    |   movel([0.131422, -1.358046, -2.590069, -0.764274, 1.570796, 1.702219],accel_mss,speed_ms,0,blend_radius_m)
    |   movel([0.131217, -1.358381, -2.589844, -0.764164, 1.570796, 1.702013],accel_mss,speed_ms,0,blend_radius_m)
    |   movel([0.131469, -1.358672, -2.589647, -0.764069, 1.570796, 1.702265],accel_mss,speed_ms,0,blend_radius_m)
    |   movel([0.131675, -1.358796, -2.589564, -0.764029, 1.570796, 1.702471],accel_mss,speed_ms,0,blend_radius_m)
    |   movel([0.131656, -1.359066, -2.589382, -0.763941, 1.570796, 1.702453],accel_mss,speed_ms,0,blend_radius_m)
    |   movel([0.131428, -1.359319, -2.589211, -0.763858, 1.570796, 1.702225],accel_mss,speed_ms,0,blend_radius_m)
    |   movel([0.131132, -1.359619, -2.589009, -0.763761, 1.570796, 1.701929],accel_mss,speed_ms,0,blend_radius_m)
    |   movel([0.127085, -1.360149, -2.588651, -0.763589, 1.570796, 1.697882],accel_mss,speed_ms,0,blend_radius_m)
    |   movel([0.125499, -1.360363, -2.588507, -0.763519, 1.570796, 1.696296],accel_mss,speed_ms,0,blend_radius_m)
    |   movel([0.124079, -1.360556, -2.588376, -0.763457, 1.570796, 1.694875],accel_mss,speed_ms,0,blend_radius_m)
    |   movel([0.122882, -1.360722, -2.588264, -0.763403, 1.570796, 1.693678],accel_mss,speed_ms,0,blend_radius_m)
    |   movel([0.122534, -1.360775, -2.588228, -0.763386, 1.570796, 1.693331],accel_mss,speed_ms,0,blend_radius_m)
    |   movel([0.122267, -1.360818, -2.588199, -0.763372, 1.570796, 1.693063],accel_mss,speed_ms,0,blend_radius_m)
    |   movel([0.121847, -1.360878, -2.588158, -0.763353, 1.570796, 1.692643],accel_mss,speed_ms,0,blend_radius_m)
    |   movel([0.121369, -1.360945, -2.588113, -0.763331, 1.570796, 1.692165],accel_mss,speed_ms,0,blend_radius_m)
    |   movel([0.120899, -1.361009, -2.588070, -0.763311, 1.570796, 1.691695],accel_mss,speed_ms,0,blend_radius_m)
    |   movel([0.120401, -1.361077, -2.588023, -0.763288, 1.570796, 1.691197],accel_mss,speed_ms,0,blend_radius_m)
    |   movel([0.119840, -1.361153, -2.587972, -0.763264, 1.570796, 1.690636],accel_mss,speed_ms,0,blend_radius_m)
    |   movel([0.119304, -1.361228, -2.587921, -0.763240, 1.570796, 1.690101],accel_mss,speed_ms,0,blend_radius_m)
    |   movel([0.118887, -1.361287, -2.587881, -0.763221, 1.570796, 1.689683],accel_mss,speed_ms,0,blend_radius_m)
    |   movel([0.118469, -1.361347, -2.587840, -0.763201, 1.570796, 1.689265],accel_mss,speed_ms,0,blend_radius_m)
    |   movel([0.117933, -1.361421, -2.587790, -0.763178, 1.570796, 1.688730],accel_mss,speed_ms,0,blend_radius_m)
    |   movel([0.117372, -1.361500, -2.587737, -0.763152, 1.570796, 1.688169],accel_mss,speed_ms,0,blend_radius_m)
    |   movel([0.116874, -1.361570, -2.587689, -0.763129, 1.570796, 1.687671],accel_mss,speed_ms,0,blend_radius_m)
    |   movel([0.114544, -1.361902, -2.587464, -0.763022, 1.570796, 1.685341],accel_mss,speed_ms,0,blend_radius_m)
    |   movel([0.111844, -1.362308, -2.587189, -0.762892, 1.570796, 1.682641],accel_mss,speed_ms,0,blend_radius_m)
    |   movel([0.109120, -1.362733, -2.586901, -0.762756, 1.570796, 1.679916],accel_mss,speed_ms,0,blend_radius_m)
    |   movel([0.108772, -1.362809, -2.586848, -0.762731, 1.570796, 1.679568],accel_mss,speed_ms,0,blend_radius_m)
    |   movel([0.108514, -1.362574, -2.587008, -0.762807, 1.570796, 1.679311],accel_mss,speed_ms,0,blend_radius_m)
    |   movel([0.108672, -1.362243, -2.587233, -0.762913, 1.570796, 1.679468],accel_mss,speed_ms,0,blend_radius_m)
    |   movel([0.108981, -1.361907, -2.587461, -0.763021, 1.570796, 1.679777],accel_mss,speed_ms,0,blend_radius_m)
    |   movel([0.109311, -1.361648, -2.587636, -0.763104, 1.570796, 1.680107],accel_mss,speed_ms,0,blend_radius_m)
    |   movel([0.109605, -1.361472, -2.587756, -0.763161, 1.570796, 1.680401],accel_mss,speed_ms,0,blend_radius_m)
    |   movel([0.109666, -1.361181, -2.587953, -0.763255, 1.570796, 1.680463],accel_mss,speed_ms,0,blend_radius_m)
    |   movel([0.109470, -1.361072, -2.588027, -0.763290, 1.570796, 1.680266],accel_mss,speed_ms,0,blend_radius_m)
    |   movel([0.109530, -1.360833, -2.588189, -0.763367, 1.570796, 1.680326],accel_mss,speed_ms,0,blend_radius_m)
    |   movel([0.109705, -1.360578, -2.588361, -0.763450, 1.570796, 1.680502],accel_mss,speed_ms,0,blend_radius_m)
    |   movel([0.109652, -1.360212, -2.588608, -0.763568, 1.570796, 1.680449],accel_mss,speed_ms,0,blend_radius_m)
    |   movel([0.109837, -1.359966, -2.588775, -0.763648, 1.570796, 1.680633],accel_mss,speed_ms,0,blend_radius_m)
    |   movel([0.109967, -1.359524, -2.589073, -0.763792, 1.570796, 1.680764],accel_mss,speed_ms,0,blend_radius_m)
    |   movel([0.110006, -1.359241, -2.589264, -0.763884, 1.570796, 1.680802],accel_mss,speed_ms,0,blend_radius_m)
    |   movel([0.110093, -1.358670, -2.589649, -0.764070, 1.570796, 1.680889],accel_mss,speed_ms,0,blend_radius_m)
    |   movel([0.110206, -1.358204, -2.589963, -0.764222, 1.570796, 1.681003],accel_mss,speed_ms,0,blend_radius_m)
    |   movel([0.110408, -1.357592, -2.590375, -0.764422, 1.570796, 1.681205],accel_mss,speed_ms,0,blend_radius_m)
    |   movel([0.110894, -1.356270, -2.591262, -0.764857, 1.570796, 1.681691],accel_mss,speed_ms,0,blend_radius_m)
    |   movel([0.111101, -1.355724, -2.591628, -0.765037, 1.570796, 1.681897],accel_mss,speed_ms,0,blend_radius_m)
    |   movel([0.111293, -1.355253, -2.591943, -0.765193, 1.570796, 1.682089],accel_mss,speed_ms,0,blend_radius_m)
    |   movel([0.111466, -1.354854, -2.592210, -0.765325, 1.570796, 1.682262],accel_mss,speed_ms,0,blend_radius_m)
    |   movel([0.111570, -1.354589, -2.592387, -0.765413, 1.570796, 1.682366],accel_mss,speed_ms,0,blend_radius_m)
    |   movel([0.111744, -1.354339, -2.592554, -0.765496, 1.570796, 1.682540],accel_mss,speed_ms,0,blend_radius_m)
    |   movel([0.111777, -1.353985, -2.592790, -0.765614, 1.570796, 1.682573],accel_mss,speed_ms,0,blend_radius_m)
    |   movel([0.112301, -1.352877, -2.593529, -0.765984, 1.570796, 1.683097],accel_mss,speed_ms,0,blend_radius_m)
    |   movel([0.112851, -1.351791, -2.594251, -0.766348, 1.570796, 1.683647],accel_mss,speed_ms,0,blend_radius_m)
    |   movel([0.113284, -1.351070, -2.594729, -0.766590, 1.570796, 1.684081],accel_mss,speed_ms,0,blend_radius_m)
    |   movel([0.113462, -1.350817, -2.594896, -0.766675, 1.570796, 1.684258],accel_mss,speed_ms,0,blend_radius_m)
    |   movel([0.113667, -1.350551, -2.595073, -0.766765, 1.570796, 1.684463],accel_mss,speed_ms,0,blend_radius_m)
    |   movel([0.113872, -1.350302, -2.595238, -0.766849, 1.570796, 1.684668],accel_mss,speed_ms,0,blend_radius_m)
    |   movel([0.114255, -1.349877, -2.595519, -0.766993, 1.570796, 1.685052],accel_mss,speed_ms,0,blend_radius_m)
    |   movel([0.114419, -1.349522, -2.595753, -0.767113, 1.570796, 1.685216],accel_mss,speed_ms,0,blend_radius_m)
    |   movel([0.114172, -1.349540, -2.595742, -0.767107, 1.570796, 1.684968],accel_mss,speed_ms,0,blend_radius_m)
    |   movel([0.113906, -1.349563, -2.595727, -0.767099, 1.570796, 1.684702],accel_mss,speed_ms,0,blend_radius_m)
    |   movel([0.113638, -1.349488, -2.595776, -0.767125, 1.570796, 1.684434],accel_mss,speed_ms,0,blend_radius_m)
    |   movel([0.113581, -1.349115, -2.596022, -0.767251, 1.570796, 1.684377],accel_mss,speed_ms,0,blend_radius_m)
    |   movel([0.113640, -1.348716, -2.596286, -0.767387, 1.570796, 1.684437],accel_mss,speed_ms,0,blend_radius_m)
    |   movel([0.113813, -1.348451, -2.596461, -0.767477, 1.570796, 1.684609],accel_mss,speed_ms,0,blend_radius_m)
    |   movel([0.114104, -1.348214, -2.596617, -0.767558, 1.570796, 1.684901],accel_mss,speed_ms,0,blend_radius_m)
    |   movel([0.114427, -1.348012, -2.596750, -0.767627, 1.570796, 1.685223],accel_mss,speed_ms,0,blend_radius_m)
    |   movel([0.114780, -1.347843, -2.596862, -0.767685, 1.570796, 1.685576],accel_mss,speed_ms,0,blend_radius_m)
    |   movel([0.115153, -1.347715, -2.596946, -0.767728, 1.570796, 1.685950],accel_mss,speed_ms,0,blend_radius_m)
    |   movel([0.115538, -1.347574, -2.597038, -0.767776, 1.570796, 1.686334],accel_mss,speed_ms,0,blend_radius_m)
    |   movel([0.116178, -1.347179, -2.597299, -0.767912, 1.570796, 1.686974],accel_mss,speed_ms,0,blend_radius_m)
    |   movel([0.118416, -1.346430, -2.597791, -0.768168, 1.570796, 1.689213],accel_mss,speed_ms,0,blend_radius_m)
    |   movel([0.120675, -1.345699, -2.598271, -0.768420, 1.570796, 1.691471],accel_mss,speed_ms,0,blend_radius_m)
    |   movel([0.120996, -1.345719, -2.598257, -0.768413, 1.570796, 1.691792],accel_mss,speed_ms,0,blend_radius_m)
    |   movel([0.121352, -1.345738, -2.598245, -0.768406, 1.570796, 1.692148],accel_mss,speed_ms,0,blend_radius_m)
    |   movel([0.121691, -1.345520, -2.598388, -0.768481, 1.570796, 1.692487],accel_mss,speed_ms,0,blend_radius_m)
    |   movel([0.121589, -1.345278, -2.598546, -0.768565, 1.570796, 1.692385],accel_mss,speed_ms,0,blend_radius_m)
    |   movel([0.121500, -1.344976, -2.598744, -0.768669, 1.570796, 1.692296],accel_mss,speed_ms,0,blend_radius_m)
    |   movel([0.121695, -1.344748, -2.598893, -0.768748, 1.570796, 1.692491],accel_mss,speed_ms,0,blend_radius_m)
    |   movel([0.122038, -1.344499, -2.599056, -0.768834, 1.570796, 1.692835],accel_mss,speed_ms,0,blend_radius_m)
    |   movel([0.122298, -1.344313, -2.599178, -0.768898, 1.570796, 1.693094],accel_mss,speed_ms,0,blend_radius_m)
    |   movel([0.122428, -1.344051, -2.599349, -0.768989, 1.570796, 1.693224],accel_mss,speed_ms,0,blend_radius_m)
    |   movel([0.122134, -1.344045, -2.599353, -0.768991, 1.570796, 1.692931],accel_mss,speed_ms,0,blend_radius_m)
    |   movel([0.121865, -1.344049, -2.599350, -0.768989, 1.570796, 1.692661],accel_mss,speed_ms,0,blend_radius_m)
    |   movel([0.121926, -1.343536, -2.599686, -0.769168, 1.570796, 1.692722],accel_mss,speed_ms,0,blend_radius_m)
    |   movel([0.122108, -1.342970, -2.600055, -0.769365, 1.570796, 1.692904],accel_mss,speed_ms,0,blend_radius_m)
    |   movel([0.122198, -1.342705, -2.600227, -0.769457, 1.570796, 1.692994],accel_mss,speed_ms,0,blend_radius_m)
    |   movel([0.122277, -1.342458, -2.600388, -0.769543, 1.570796, 1.693074],accel_mss,speed_ms,0,blend_radius_m)
    |   movel([0.122367, -1.342155, -2.600585, -0.769649, 1.570796, 1.693164],accel_mss,speed_ms,0,blend_radius_m)
    |   movel([0.122577, -1.341845, -2.600787, -0.769757, 1.570796, 1.693373],accel_mss,speed_ms,0,blend_radius_m)
    |   movel([0.122789, -1.341589, -2.600953, -0.769846, 1.570796, 1.693585],accel_mss,speed_ms,0,blend_radius_m)
    |   movel([0.123034, -1.341314, -2.601133, -0.769943, 1.570796, 1.693831],accel_mss,speed_ms,0,blend_radius_m)
    |   movel([0.123671, -1.340622, -2.601581, -0.770185, 1.570796, 1.694467],accel_mss,speed_ms,0,blend_radius_m)
    |   movel([0.124629, -1.340427, -2.601708, -0.770254, 1.570796, 1.695426],accel_mss,speed_ms,0,blend_radius_m)
    |   movel([0.125882, -1.340203, -2.601853, -0.770333, 1.570796, 1.696678],accel_mss,speed_ms,0,blend_radius_m)
    |   movel([0.127200, -1.340030, -2.601965, -0.770394, 1.570796, 1.697996],accel_mss,speed_ms,0,blend_radius_m)
    |   movel([0.128376, -1.339917, -2.602039, -0.770434, 1.570796, 1.699172],accel_mss,speed_ms,0,blend_radius_m)
    |   movel([0.128803, -1.339961, -2.602010, -0.770418, 1.570796, 1.699599],accel_mss,speed_ms,0,blend_radius_m)
    |   movel([0.129089, -1.340087, -2.601928, -0.770374, 1.570796, 1.699886],accel_mss,speed_ms,0,blend_radius_m)
    |   movel([0.129309, -1.340254, -2.601820, -0.770315, 1.570796, 1.700106],accel_mss,speed_ms,0,blend_radius_m)
    |   movel([0.129435, -1.340429, -2.601707, -0.770253, 1.570796, 1.700231],accel_mss,speed_ms,0,blend_radius_m)
    |   movel([0.129396, -1.340689, -2.601538, -0.770162, 1.570796, 1.700193],accel_mss,speed_ms,0,blend_radius_m)
    |   movel([0.129524, -1.340866, -2.601423, -0.770100, 1.570796, 1.700320],accel_mss,speed_ms,0,blend_radius_m)
    |   movel([0.129472, -1.341183, -2.601217, -0.769989, 1.570796, 1.700269],accel_mss,speed_ms,0,blend_radius_m)
    |   movel([0.129264, -1.341421, -2.601063, -0.769905, 1.570796, 1.700060],accel_mss,speed_ms,0,blend_radius_m)
    |   movel([0.129247, -1.341706, -2.600878, -0.769806, 1.570796, 1.700043],accel_mss,speed_ms,0,blend_radius_m)
    |   movel([0.129226, -1.342103, -2.600619, -0.769667, 1.570796, 1.700023],accel_mss,speed_ms,0,blend_radius_m)
    |   movel([0.129118, -1.342564, -2.600319, -0.769506, 1.570796, 1.699915],accel_mss,speed_ms,0,blend_radius_m)
    |   movel([0.128966, -1.342955, -2.600064, -0.769370, 1.570796, 1.699762],accel_mss,speed_ms,0,blend_radius_m)
    |   movel([0.128664, -1.343092, -2.599975, -0.769322, 1.570796, 1.699461],accel_mss,speed_ms,0,blend_radius_m)
    |   movel([0.128382, -1.343292, -2.599845, -0.769252, 1.570796, 1.699178],accel_mss,speed_ms,0,blend_radius_m)
    |   movel([0.128379, -1.343588, -2.599652, -0.769150, 1.570796, 1.699175],accel_mss,speed_ms,0,blend_radius_m)
    |   movel([0.128483, -1.343834, -2.599491, -0.769064, 1.570796, 1.699279],accel_mss,speed_ms,0,blend_radius_m)
    |   movel([0.128519, -1.344124, -2.599301, -0.768964, 1.570796, 1.699315],accel_mss,speed_ms,0,blend_radius_m)
    |   movel([0.128237, -1.344388, -2.599129, -0.768872, 1.570796, 1.699033],accel_mss,speed_ms,0,blend_radius_m)
    |   movel([0.128151, -1.344682, -2.598937, -0.768771, 1.570796, 1.698948],accel_mss,speed_ms,0,blend_radius_m)
    |   movel([0.128545, -1.344644, -2.598961, -0.768784, 1.570796, 1.699342],accel_mss,speed_ms,0,blend_radius_m)
    |   movel([0.129417, -1.344531, -2.599035, -0.768823, 1.570796, 1.700213],accel_mss,speed_ms,0,blend_radius_m)
    |   movel([0.130216, -1.344512, -2.599048, -0.768829, 1.570796, 1.701013],accel_mss,speed_ms,0,blend_radius_m)
    |   movel([0.130962, -1.344536, -2.599032, -0.768821, 1.570796, 1.701758],accel_mss,speed_ms,0,blend_radius_m)
    |   movel([0.131239, -1.344625, -2.598974, -0.768790, 1.570796, 1.702036],accel_mss,speed_ms,0,blend_radius_m)
    |   movel([0.131699, -1.344650, -2.598957, -0.768781, 1.570796, 1.702495],accel_mss,speed_ms,0,blend_radius_m)
    |   movel([0.132047, -1.344467, -2.599077, -0.768845, 1.570796, 1.702843],accel_mss,speed_ms,0,blend_radius_m)
    |   movel([0.131918, -1.344291, -2.599192, -0.768906, 1.570796, 1.702714],accel_mss,speed_ms,0,blend_radius_m)
    |   movel([0.131651, -1.344100, -2.599317, -0.768972, 1.570796, 1.702447],accel_mss,speed_ms,0,blend_radius_m)
    |   movel([0.132106, -1.343657, -2.599607, -0.769126, 1.570796, 1.702902],accel_mss,speed_ms,0,blend_radius_m)
    |   movel([0.132430, -1.343451, -2.599741, -0.769197, 1.570796, 1.703227],accel_mss,speed_ms,0,blend_radius_m)
    |   movel([0.132572, -1.343210, -2.599898, -0.769281, 1.570796, 1.703368],accel_mss,speed_ms,0,blend_radius_m)
    |   movel([0.132296, -1.343074, -2.599987, -0.769328, 1.570796, 1.703093],accel_mss,speed_ms,0,blend_radius_m)
    |   movel([0.132431, -1.342597, -2.600298, -0.769494, 1.570796, 1.703227],accel_mss,speed_ms,0,blend_radius_m)
    |   movel([0.132665, -1.342355, -2.600455, -0.769579, 1.570796, 1.703462],accel_mss,speed_ms,0,blend_radius_m)
    |   movel([0.133142, -1.342023, -2.600671, -0.769695, 1.570796, 1.703938],accel_mss,speed_ms,0,blend_radius_m)
    |   movel([0.133515, -1.341866, -2.600774, -0.769750, 1.570796, 1.704311],accel_mss,speed_ms,0,blend_radius_m)
    |   movel([0.133874, -1.341846, -2.600787, -0.769757, 1.570796, 1.704671],accel_mss,speed_ms,0,blend_radius_m)
    |   movel([0.134312, -1.341959, -2.600713, -0.769717, 1.570796, 1.705108],accel_mss,speed_ms,0,blend_radius_m)
    |   movel([0.134537, -1.342047, -2.600656, -0.769686, 1.570796, 1.705333],accel_mss,speed_ms,0,blend_radius_m)
    |   movel([0.134724, -1.342134, -2.600599, -0.769656, 1.570796, 1.705520],accel_mss,speed_ms,0,blend_radius_m)
    |   movel([0.134889, -1.342254, -2.600521, -0.769614, 1.570796, 1.705685],accel_mss,speed_ms,0,blend_radius_m)
    |   movel([0.135058, -1.342462, -2.600386, -0.769541, 1.570796, 1.705854],accel_mss,speed_ms,0,blend_radius_m)
    |   movel([0.135120, -1.342790, -2.600172, -0.769427, 1.570796, 1.705917],accel_mss,speed_ms,0,blend_radius_m)
    |   movel([0.134596, -1.343303, -2.599837, -0.769249, 1.570796, 1.705392],accel_mss,speed_ms,0,blend_radius_m)
    |   movel([0.134152, -1.343634, -2.599621, -0.769134, 1.570796, 1.704948],accel_mss,speed_ms,0,blend_radius_m)
    |   movel([0.134394, -1.343806, -2.599509, -0.769074, 1.570796, 1.705190],accel_mss,speed_ms,0,blend_radius_m)
    |   movel([0.134638, -1.343980, -2.599395, -0.769013, 1.570796, 1.705434],accel_mss,speed_ms,0,blend_radius_m)
    |   movel([0.134303, -1.344283, -2.599197, -0.768908, 1.570796, 1.705100],accel_mss,speed_ms,0,blend_radius_m)
    |   movel([0.133995, -1.344518, -2.599044, -0.768827, 1.570796, 1.704791],accel_mss,speed_ms,0,blend_radius_m)
    |   movel([0.133724, -1.344655, -2.598954, -0.768780, 1.570796, 1.704520],accel_mss,speed_ms,0,blend_radius_m)
    |   movel([0.133806, -1.344937, -2.598770, -0.768682, 1.570796, 1.704602],accel_mss,speed_ms,0,blend_radius_m)
    |   movel([0.134102, -1.344945, -2.598764, -0.768679, 1.570796, 1.704899],accel_mss,speed_ms,0,blend_radius_m)
    |   movel([0.134405, -1.344992, -2.598733, -0.768663, 1.570796, 1.705202],accel_mss,speed_ms,0,blend_radius_m)
    |   movel([0.134632, -1.345146, -2.598633, -0.768610, 1.570796, 1.705428],accel_mss,speed_ms,0,blend_radius_m)
    |   movel([0.134781, -1.345283, -2.598543, -0.768563, 1.570796, 1.705577],accel_mss,speed_ms,0,blend_radius_m)
    |   movel([0.134990, -1.345391, -2.598472, -0.768526, 1.570796, 1.705786],accel_mss,speed_ms,0,blend_radius_m)
    |   movel([0.134941, -1.345692, -2.598275, -0.768422, 1.570796, 1.705737],accel_mss,speed_ms,0,blend_radius_m)
    |   movel([0.134735, -1.345909, -2.598133, -0.768347, 1.570796, 1.705532],accel_mss,speed_ms,0,blend_radius_m)
    |   movel([0.134593, -1.346186, -2.597951, -0.768252, 1.570796, 1.705389],accel_mss,speed_ms,0,blend_radius_m)
    |   movel([0.134351, -1.346477, -2.597760, -0.768152, 1.570796, 1.705148],accel_mss,speed_ms,0,blend_radius_m)
    |   movel([0.134008, -1.346695, -2.597616, -0.768077, 1.570796, 1.704805],accel_mss,speed_ms,0,blend_radius_m)
    |   movel([0.133511, -1.346849, -2.597515, -0.768024, 1.570796, 1.704307],accel_mss,speed_ms,0,blend_radius_m)
    |   speed_ms = 0.003
    |   movel([0.133372, -1.333561, -2.591198, -0.787631, 1.570796, 1.704169],accel_mss,speed_ms,0,blend_radius_m)
    |   speed_ms = 1.000
    |   movel([0.133372, -1.307920, -2.578330, -0.826139, 1.570796, 1.704169],accel_mss,speed_ms,0,blend_radius_m)
    |   movel([0.124146, -1.335219, -2.560894, -0.816276, 1.570796, 1.694943],accel_mss,speed_ms,0,blend_radius_m)
    |   movel([0.124146, -1.360403, -2.573410, -0.778576, 1.570796, 1.694943],accel_mss,speed_ms,0,blend_radius_m)
    |   speed_ms = 0.003
    |   movel([0.124146, -1.370225, -2.577968, -0.764196, 1.570796, 1.694943],accel_mss,speed_ms,0,blend_radius_m)
    |   speed_ms = 0.007
    |   movel([0.123793, -1.371087, -2.577372, -0.763930, 1.570796, 1.694589],accel_mss,speed_ms,0,blend_radius_m)
    |   movel([0.123280, -1.371916, -2.576797, -0.763676, 1.570796, 1.694077],accel_mss,speed_ms,0,blend_radius_m)
    |   movel([0.122665, -1.372875, -2.576132, -0.763382, 1.570796, 1.693461],accel_mss,speed_ms,0,blend_radius_m)
    |   movel([0.121838, -1.374160, -2.575237, -0.762992, 1.570796, 1.692634],accel_mss,speed_ms,0,blend_radius_m)
    |   movel([0.121407, -1.374875, -2.574738, -0.762775, 1.570796, 1.692203],accel_mss,speed_ms,0,blend_radius_m)
    |   movel([0.121174, -1.375318, -2.574429, -0.762642, 1.570796, 1.691970],accel_mss,speed_ms,0,blend_radius_m)
    |   movel([0.121312, -1.375503, -2.574300, -0.762586, 1.570796, 1.692108],accel_mss,speed_ms,0,blend_radius_m)
    |   movel([0.121589, -1.375475, -2.574320, -0.762595, 1.570796, 1.692385],accel_mss,speed_ms,0,blend_radius_m)
    |   movel([0.122025, -1.375385, -2.574382, -0.762621, 1.570796, 1.692821],accel_mss,speed_ms,0,blend_radius_m)
    |   movel([0.122716, -1.375209, -2.574505, -0.762675, 1.570796, 1.693512],accel_mss,speed_ms,0,blend_radius_m)
    |   movel([0.123641, -1.374975, -2.574669, -0.762745, 1.570796, 1.694437],accel_mss,speed_ms,0,blend_radius_m)
    |   movel([0.124044, -1.374911, -2.574713, -0.762764, 1.570796, 1.694840],accel_mss,speed_ms,0,blend_radius_m)
    |   movel([0.124195, -1.375102, -2.574580, -0.762707, 1.570796, 1.694992],accel_mss,speed_ms,0,blend_radius_m)
    |   movel([0.123079, -1.376507, -2.573598, -0.762284, 1.570796, 1.693875],accel_mss,speed_ms,0,blend_radius_m)
    |   movel([0.121902, -1.377963, -2.572577, -0.761849, 1.570796, 1.692699],accel_mss,speed_ms,0,blend_radius_m)
    |   movel([0.120523, -1.379657, -2.571385, -0.761347, 1.570796, 1.691319],accel_mss,speed_ms,0,blend_radius_m)
    |   movel([0.119131, -1.381360, -2.570183, -0.760846, 1.570796, 1.689928],accel_mss,speed_ms,0,blend_radius_m)
    |   movel([0.117908, -1.382848, -2.569129, -0.760412, 1.570796, 1.688704],accel_mss,speed_ms,0,blend_radius_m)
    |   movel([0.116864, -1.384114, -2.568230, -0.760045, 1.570796, 1.687661],accel_mss,speed_ms,0,blend_radius_m)
    |   movel([0.116633, -1.384373, -2.568045, -0.759971, 1.570796, 1.687429],accel_mss,speed_ms,0,blend_radius_m)
    |   movel([0.116427, -1.384584, -2.567895, -0.759910, 1.570796, 1.687224],accel_mss,speed_ms,0,blend_radius_m)
    |   movel([0.116381, -1.384342, -2.568068, -0.759980, 1.570796, 1.687177],accel_mss,speed_ms,0,blend_radius_m)
    |   movel([0.116785, -1.383473, -2.568685, -0.760231, 1.570796, 1.687582],accel_mss,speed_ms,0,blend_radius_m)
    |   movel([0.117268, -1.382455, -2.569408, -0.760527, 1.570796, 1.688064],accel_mss,speed_ms,0,blend_radius_m)
    |   movel([0.117834, -1.381287, -2.570234, -0.760868, 1.570796, 1.688631],accel_mss,speed_ms,0,blend_radius_m)
    |   movel([0.118529, -1.379857, -2.571244, -0.761288, 1.570796, 1.689326],accel_mss,speed_ms,0,blend_radius_m)
    |   movel([0.118953, -1.378940, -2.571890, -0.761559, 1.570796, 1.689749],accel_mss,speed_ms,0,blend_radius_m)
    |   movel([0.119224, -1.378300, -2.572340, -0.761749, 1.570796, 1.690020],accel_mss,speed_ms,0,blend_radius_m)
    |   movel([0.119087, -1.378136, -2.572455, -0.761798, 1.570796, 1.689884],accel_mss,speed_ms,0,blend_radius_m)
    |   movel([0.118747, -1.378188, -2.572418, -0.761782, 1.570796, 1.689544],accel_mss,speed_ms,0,blend_radius_m)
    |   movel([0.118246, -1.378296, -2.572343, -0.761750, 1.570796, 1.689042],accel_mss,speed_ms,0,blend_radius_m)
    |   movel([0.117501, -1.378488, -2.572208, -0.761693, 1.570796, 1.688298],accel_mss,speed_ms,0,blend_radius_m)
    |   movel([0.116757, -1.378680, -2.572073, -0.761636, 1.570796, 1.687553],accel_mss,speed_ms,0,blend_radius_m)
    |   movel([0.116258, -1.378787, -2.571997, -0.761604, 1.570796, 1.687054],accel_mss,speed_ms,0,blend_radius_m)
    |   movel([0.115918, -1.378840, -2.571960, -0.761589, 1.570796, 1.686714],accel_mss,speed_ms,0,blend_radius_m)
    |   movel([0.115788, -1.378677, -2.572075, -0.761637, 1.570796, 1.686584],accel_mss,speed_ms,0,blend_radius_m)
    |   movel([0.116123, -1.377916, -2.572609, -0.761863, 1.570796, 1.686920],accel_mss,speed_ms,0,blend_radius_m)
    |   movel([0.116612, -1.376865, -2.573347, -0.762177, 1.570796, 1.687408],accel_mss,speed_ms,0,blend_radius_m)
    |   movel([0.117386, -1.375283, -2.574453, -0.762652, 1.570796, 1.688182],accel_mss,speed_ms,0,blend_radius_m)
    |   movel([0.118051, -1.373950, -2.575383, -0.763055, 1.570796, 1.688847],accel_mss,speed_ms,0,blend_radius_m)
    |   movel([0.118642, -1.372791, -2.576190, -0.763408, 1.570796, 1.689439],accel_mss,speed_ms,0,blend_radius_m)
    |   movel([0.119160, -1.371793, -2.576883, -0.763713, 1.570796, 1.689956],accel_mss,speed_ms,0,blend_radius_m)
    |   movel([0.119467, -1.371483, -2.577098, -0.763808, 1.570796, 1.690263],accel_mss,speed_ms,0,blend_radius_m)
    |   movel([0.119865, -1.371330, -2.577204, -0.763855, 1.570796, 1.690661],accel_mss,speed_ms,0,blend_radius_m)
    |   movel([0.120531, -1.371128, -2.577343, -0.763917, 1.570796, 1.691328],accel_mss,speed_ms,0,blend_radius_m)
    |   movel([0.121831, -1.370775, -2.577588, -0.764026, 1.570796, 1.692628],accel_mss,speed_ms,0,blend_radius_m)
    |   movel([0.122994, -1.370473, -2.577797, -0.764119, 1.570796, 1.693790],accel_mss,speed_ms,0,blend_radius_m)
    |   movel([0.123692, -1.370311, -2.577909, -0.764169, 1.570796, 1.694488],accel_mss,speed_ms,0,blend_radius_m)
    |   movel([0.124146, -1.370225, -2.577968, -0.764196, 1.570796, 1.694943],accel_mss,speed_ms,0,blend_radius_m)
    |   speed_ms = 0.003
    |   movel([0.124146, -1.373545, -2.579471, -0.759372, 1.570796, 1.694943],accel_mss,speed_ms,0,blend_radius_m)
    |   speed_ms = 0.007
    |   movel([0.123793, -1.374405, -2.578873, -0.759111, 1.570796, 1.694589],accel_mss,speed_ms,0,blend_radius_m)
    |   movel([0.123280, -1.375232, -2.578297, -0.758860, 1.570796, 1.694077],accel_mss,speed_ms,0,blend_radius_m)
    |   movel([0.122665, -1.376188, -2.577630, -0.758571, 1.570796, 1.693461],accel_mss,speed_ms,0,blend_radius_m)
    |   movel([0.121838, -1.377470, -2.576733, -0.758186, 1.570796, 1.692634],accel_mss,speed_ms,0,blend_radius_m)
    |   movel([0.121407, -1.378183, -2.576233, -0.757972, 1.570796, 1.692203],accel_mss,speed_ms,0,blend_radius_m)
    |   movel([0.121174, -1.378625, -2.575924, -0.757841, 1.570796, 1.691970],accel_mss,speed_ms,0,blend_radius_m)
    |   movel([0.121312, -1.378810, -2.575794, -0.757786, 1.570796, 1.692108],accel_mss,speed_ms,0,blend_radius_m)
    |   movel([0.121589, -1.378781, -2.575814, -0.757794, 1.570796, 1.692385],accel_mss,speed_ms,0,blend_radius_m)
    |   movel([0.122025, -1.378692, -2.575877, -0.757821, 1.570796, 1.692821],accel_mss,speed_ms,0,blend_radius_m)
    |   movel([0.122716, -1.378516, -2.576000, -0.757873, 1.570796, 1.693512],accel_mss,speed_ms,0,blend_radius_m)
    |   movel([0.123641, -1.378282, -2.576164, -0.757943, 1.570796, 1.694437],accel_mss,speed_ms,0,blend_radius_m)
    |   movel([0.124044, -1.378219, -2.576208, -0.757962, 1.570796, 1.694840],accel_mss,speed_ms,0,blend_radius_m)
    |   movel([0.124195, -1.378409, -2.576075, -0.757905, 1.570796, 1.694992],accel_mss,speed_ms,0,blend_radius_m)
    |   movel([0.123079, -1.379810, -2.575090, -0.757489, 1.570796, 1.693875],accel_mss,speed_ms,0,blend_radius_m)
    |   movel([0.121902, -1.381262, -2.574067, -0.757060, 1.570796, 1.692699],accel_mss,speed_ms,0,blend_radius_m)
    |   movel([0.120523, -1.382952, -2.572872, -0.756565, 1.570796, 1.691319],accel_mss,speed_ms,0,blend_radius_m)
    |   movel([0.119131, -1.384650, -2.571667, -0.756072, 1.570796, 1.689928],accel_mss,speed_ms,0,blend_radius_m)
    |   movel([0.117908, -1.386135, -2.570610, -0.755644, 1.570796, 1.688704],accel_mss,speed_ms,0,blend_radius_m)
    |   movel([0.116864, -1.387397, -2.569710, -0.755283, 1.570796, 1.687661],accel_mss,speed_ms,0,blend_radius_m)
    |   movel([0.116633, -1.387655, -2.569525, -0.755209, 1.570796, 1.687429],accel_mss,speed_ms,0,blend_radius_m)
    |   movel([0.116427, -1.387865, -2.569374, -0.755149, 1.570796, 1.687224],accel_mss,speed_ms,0,blend_radius_m)
    |   movel([0.116381, -1.387624, -2.569547, -0.755218, 1.570796, 1.687177],accel_mss,speed_ms,0,blend_radius_m)
    |   movel([0.116785, -1.386757, -2.570166, -0.755465, 1.570796, 1.687582],accel_mss,speed_ms,0,blend_radius_m)
    |   movel([0.117268, -1.385742, -2.570890, -0.755757, 1.570796, 1.688064],accel_mss,speed_ms,0,blend_radius_m)
    |   movel([0.117834, -1.384578, -2.571719, -0.756093, 1.570796, 1.688631],accel_mss,speed_ms,0,blend_radius_m)
    |   movel([0.118529, -1.383151, -2.572731, -0.756507, 1.570796, 1.689326],accel_mss,speed_ms,0,blend_radius_m)
    |   movel([0.118953, -1.382237, -2.573378, -0.756774, 1.570796, 1.689749],accel_mss,speed_ms,0,blend_radius_m)
    |   movel([0.119224, -1.381599, -2.573829, -0.756961, 1.570796, 1.690020],accel_mss,speed_ms,0,blend_radius_m)
    |   movel([0.119087, -1.381435, -2.573945, -0.757009, 1.570796, 1.689884],accel_mss,speed_ms,0,blend_radius_m)
    |   movel([0.118747, -1.381487, -2.573908, -0.756994, 1.570796, 1.689544],accel_mss,speed_ms,0,blend_radius_m)
    |   movel([0.118246, -1.381595, -2.573832, -0.756962, 1.570796, 1.689042],accel_mss,speed_ms,0,blend_radius_m)
    |   movel([0.117501, -1.381786, -2.573697, -0.756906, 1.570796, 1.688298],accel_mss,speed_ms,0,blend_radius_m)
    |   movel([0.116757, -1.381977, -2.573562, -0.756850, 1.570796, 1.687553],accel_mss,speed_ms,0,blend_radius_m)
    |   movel([0.116258, -1.382085, -2.573486, -0.756818, 1.570796, 1.687054],accel_mss,speed_ms,0,blend_radius_m)
    |   movel([0.115918, -1.382138, -2.573448, -0.756803, 1.570796, 1.686714],accel_mss,speed_ms,0,blend_radius_m)
    |   movel([0.115788, -1.381975, -2.573563, -0.756851, 1.570796, 1.686584],accel_mss,speed_ms,0,blend_radius_m)
    |   movel([0.116123, -1.381216, -2.574099, -0.757073, 1.570796, 1.686920],accel_mss,speed_ms,0,blend_radius_m)
    |   movel([0.116612, -1.380167, -2.574839, -0.757383, 1.570796, 1.687408],accel_mss,speed_ms,0,blend_radius_m)
    |   movel([0.117386, -1.378590, -2.575948, -0.757851, 1.570796, 1.688182],accel_mss,speed_ms,0,blend_radius_m)
    |   movel([0.118051, -1.377261, -2.576880, -0.758248, 1.570796, 1.688847],accel_mss,speed_ms,0,blend_radius_m)
    |   movel([0.118642, -1.376105, -2.577688, -0.758596, 1.570796, 1.689439],accel_mss,speed_ms,0,blend_radius_m)
    |   movel([0.119160, -1.375109, -2.578383, -0.758897, 1.570796, 1.689956],accel_mss,speed_ms,0,blend_radius_m)
    |   movel([0.119467, -1.374800, -2.578598, -0.758991, 1.570796, 1.690263],accel_mss,speed_ms,0,blend_radius_m)
    |   movel([0.119865, -1.374647, -2.578705, -0.759037, 1.570796, 1.690661],accel_mss,speed_ms,0,blend_radius_m)
    |   movel([0.120531, -1.374446, -2.578845, -0.759098, 1.570796, 1.691328],accel_mss,speed_ms,0,blend_radius_m)
    |   movel([0.121831, -1.374094, -2.579090, -0.759205, 1.570796, 1.692628],accel_mss,speed_ms,0,blend_radius_m)
    |   movel([0.122994, -1.373793, -2.579299, -0.759297, 1.570796, 1.693790],accel_mss,speed_ms,0,blend_radius_m)
    |   movel([0.123692, -1.373631, -2.579411, -0.759346, 1.570796, 1.694488],accel_mss,speed_ms,0,blend_radius_m)
    |   movel([0.124146, -1.373545, -2.579471, -0.759372, 1.570796, 1.694943],accel_mss,speed_ms,0,blend_radius_m)
    |   speed_ms = 0.003
    |   movel([0.124146, -1.360403, -2.573410, -0.778576, 1.570796, 1.694943],accel_mss,speed_ms,0,blend_radius_m)
    |   speed_ms = 1.000
    |   movel([0.124146, -1.335219, -2.560894, -0.816276, 1.570796, 1.694943],accel_mss,speed_ms,0,blend_radius_m)
    |   movel([0.115988, -1.357886, -2.545671, -0.808832, 1.570796, 1.686785],accel_mss,speed_ms,0,blend_radius_m)
    |   movel([0.115988, -1.382667, -2.557897, -0.771824, 1.570796, 1.686785],accel_mss,speed_ms,0,blend_radius_m)
    |   speed_ms = 0.003
    |   movel([0.115988, -1.392317, -2.562347, -0.757725, 1.570796, 1.686785],accel_mss,speed_ms,0,blend_radius_m)
    |   speed_ms = 0.007
    |   movel([0.116395, -1.392329, -2.562339, -0.757721, 1.570796, 1.687191],accel_mss,speed_ms,0,blend_radius_m)
    |   movel([0.116711, -1.392556, -2.562174, -0.757658, 1.570796, 1.687507],accel_mss,speed_ms,0,blend_radius_m)
    |   movel([0.116919, -1.392985, -2.561864, -0.757540, 1.570796, 1.687715],accel_mss,speed_ms,0,blend_radius_m)
    |   movel([0.116976, -1.393318, -2.561623, -0.757448, 1.570796, 1.687772],accel_mss,speed_ms,0,blend_radius_m)
    |   movel([0.116649, -1.393630, -2.561397, -0.757362, 1.570796, 1.687445],accel_mss,speed_ms,0,blend_radius_m)
    |   movel([0.116200, -1.393658, -2.561377, -0.757355, 1.570796, 1.686996],accel_mss,speed_ms,0,blend_radius_m)
    |   movel([0.115692, -1.393625, -2.561401, -0.757364, 1.570796, 1.686488],accel_mss,speed_ms,0,blend_radius_m)
    |   movel([0.115348, -1.393521, -2.561476, -0.757392, 1.570796, 1.686144],accel_mss,speed_ms,0,blend_radius_m)
    |   movel([0.115151, -1.393344, -2.561604, -0.757441, 1.570796, 1.685947],accel_mss,speed_ms,0,blend_radius_m)
    |   movel([0.115085, -1.393091, -2.561788, -0.757511, 1.570796, 1.685881],accel_mss,speed_ms,0,blend_radius_m)
    |   movel([0.115165, -1.392773, -2.562018, -0.757598, 1.570796, 1.685962],accel_mss,speed_ms,0,blend_radius_m)
    |   movel([0.115516, -1.392508, -2.562209, -0.757672, 1.570796, 1.686313],accel_mss,speed_ms,0,blend_radius_m)
    |   movel([0.115988, -1.392317, -2.562347, -0.757725, 1.570796, 1.686785],accel_mss,speed_ms,0,blend_radius_m)
    |   speed_ms = 0.003
    |   movel([0.115988, -1.395577, -2.563814, -0.752998, 1.570796, 1.686785],accel_mss,speed_ms,0,blend_radius_m)
    |   speed_ms = 0.007
    |   movel([0.116395, -1.395589, -2.563805, -0.752995, 1.570796, 1.687191],accel_mss,speed_ms,0,blend_radius_m)
    |   movel([0.116711, -1.395816, -2.563641, -0.752933, 1.570796, 1.687507],accel_mss,speed_ms,0,blend_radius_m)
    |   movel([0.116919, -1.396243, -2.563330, -0.752816, 1.570796, 1.687715],accel_mss,speed_ms,0,blend_radius_m)
    |   movel([0.116976, -1.396576, -2.563088, -0.752726, 1.570796, 1.687772],accel_mss,speed_ms,0,blend_radius_m)
    |   movel([0.116649, -1.396886, -2.562861, -0.752641, 1.570796, 1.687445],accel_mss,speed_ms,0,blend_radius_m)
    |   movel([0.116200, -1.396914, -2.562841, -0.752634, 1.570796, 1.686996],accel_mss,speed_ms,0,blend_radius_m)
    |   movel([0.115692, -1.396881, -2.562865, -0.752643, 1.570796, 1.686488],accel_mss,speed_ms,0,blend_radius_m)
    |   movel([0.115348, -1.396778, -2.562940, -0.752671, 1.570796, 1.686144],accel_mss,speed_ms,0,blend_radius_m)
    |   movel([0.115151, -1.396601, -2.563069, -0.752719, 1.570796, 1.685947],accel_mss,speed_ms,0,blend_radius_m)
    |   movel([0.115085, -1.396349, -2.563253, -0.752787, 1.570796, 1.685881],accel_mss,speed_ms,0,blend_radius_m)
    |   movel([0.115165, -1.396032, -2.563483, -0.752874, 1.570796, 1.685962],accel_mss,speed_ms,0,blend_radius_m)
    |   movel([0.115516, -1.395768, -2.563675, -0.752946, 1.570796, 1.686313],accel_mss,speed_ms,0,blend_radius_m)
    |   movel([0.115988, -1.395577, -2.563814, -0.752998, 1.570796, 1.686785],accel_mss,speed_ms,0,blend_radius_m)
    |   speed_ms = 0.003
    |   movel([0.115988, -1.382667, -2.557897, -0.771824, 1.570796, 1.686785],accel_mss,speed_ms,0,blend_radius_m)
    |   speed_ms = 1.000
    |   movel([0.115988, -1.357886, -2.545671, -0.808832, 1.570796, 1.686785],accel_mss,speed_ms,0,blend_radius_m)
    |   movel([0.119782, -1.357452, -2.545969, -0.808968, 1.570796, 1.690578],accel_mss,speed_ms,0,blend_radius_m)
    |   movel([0.119782, -1.382241, -2.558201, -0.771947, 1.570796, 1.690578],accel_mss,speed_ms,0,blend_radius_m)
    |   speed_ms = 0.003
    |   movel([0.119782, -1.391894, -2.562653, -0.757842, 1.570796, 1.690578],accel_mss,speed_ms,0,blend_radius_m)
    |   speed_ms = 0.007
    |   movel([0.119962, -1.391564, -2.562891, -0.757933, 1.570796, 1.690759],accel_mss,speed_ms,0,blend_radius_m)
    |   movel([0.120193, -1.391304, -2.563079, -0.758006, 1.570796, 1.690989],accel_mss,speed_ms,0,blend_radius_m)
    |   movel([0.120597, -1.391186, -2.563164, -0.758039, 1.570796, 1.691393],accel_mss,speed_ms,0,blend_radius_m)
    |   movel([0.120783, -1.391316, -2.563070, -0.758003, 1.570796, 1.691579],accel_mss,speed_ms,0,blend_radius_m)
    |   movel([0.120924, -1.391495, -2.562941, -0.757953, 1.570796, 1.691720],accel_mss,speed_ms,0,blend_radius_m)
    |   movel([0.120906, -1.391791, -2.562728, -0.757871, 1.570796, 1.691703],accel_mss,speed_ms,0,blend_radius_m)
    |   movel([0.120624, -1.392181, -2.562446, -0.757762, 1.570796, 1.691420],accel_mss,speed_ms,0,blend_radius_m)
    |   movel([0.120435, -1.392385, -2.562298, -0.757706, 1.570796, 1.691231],accel_mss,speed_ms,0,blend_radius_m)
    |   movel([0.120043, -1.392729, -2.562049, -0.757611, 1.570796, 1.690839],accel_mss,speed_ms,0,blend_radius_m)
    |   movel([0.119669, -1.392658, -2.562101, -0.757630, 1.570796, 1.690465],accel_mss,speed_ms,0,blend_radius_m)
    |   movel([0.119687, -1.392232, -2.562409, -0.757748, 1.570796, 1.690484],accel_mss,speed_ms,0,blend_radius_m)
    |   movel([0.119782, -1.391894, -2.562653, -0.757842, 1.570796, 1.690578],accel_mss,speed_ms,0,blend_radius_m)
    |   speed_ms = 0.003
    |   movel([0.119782, -1.395155, -2.564120, -0.753113, 1.570796, 1.690578],accel_mss,speed_ms,0,blend_radius_m)
    |   speed_ms = 0.007
    |   movel([0.119962, -1.394827, -2.564359, -0.753203, 1.570796, 1.690759],accel_mss,speed_ms,0,blend_radius_m)
    |   movel([0.120193, -1.394568, -2.564547, -0.753275, 1.570796, 1.690989],accel_mss,speed_ms,0,blend_radius_m)
    |   movel([0.120597, -1.394450, -2.564632, -0.753307, 1.570796, 1.691393],accel_mss,speed_ms,0,blend_radius_m)
    |   movel([0.120783, -1.394579, -2.564538, -0.753271, 1.570796, 1.691579],accel_mss,speed_ms,0,blend_radius_m)
    |   movel([0.120924, -1.394757, -2.564409, -0.753222, 1.570796, 1.691720],accel_mss,speed_ms,0,blend_radius_m)
    |   movel([0.120906, -1.395052, -2.564195, -0.753141, 1.570796, 1.691703],accel_mss,speed_ms,0,blend_radius_m)
    |   movel([0.120624, -1.395442, -2.563912, -0.753035, 1.570796, 1.691420],accel_mss,speed_ms,0,blend_radius_m)
    |   movel([0.120435, -1.395645, -2.563765, -0.752979, 1.570796, 1.691231],accel_mss,speed_ms,0,blend_radius_m)
    |   movel([0.120043, -1.395988, -2.563515, -0.752886, 1.570796, 1.690839],accel_mss,speed_ms,0,blend_radius_m)
    |   movel([0.119669, -1.395917, -2.563567, -0.752905, 1.570796, 1.690465],accel_mss,speed_ms,0,blend_radius_m)
    |   movel([0.119687, -1.395493, -2.563875, -0.753021, 1.570796, 1.690484],accel_mss,speed_ms,0,blend_radius_m)
    |   movel([0.119782, -1.395155, -2.564120, -0.753113, 1.570796, 1.690578],accel_mss,speed_ms,0,blend_radius_m)
    |   speed_ms = 0.003
    |   movel([0.119782, -1.382241, -2.558201, -0.771947, 1.570796, 1.690578],accel_mss,speed_ms,0,blend_radius_m)
    |   speed_ms = 1.000
    |   movel([0.119782, -1.357452, -2.545969, -0.808968, 1.570796, 1.690578],accel_mss,speed_ms,0,blend_radius_m)
    |   movel([0.118569, -1.359477, -2.544576, -0.808336, 1.570796, 1.689365],accel_mss,speed_ms,0,blend_radius_m)
    |   movel([0.118569, -1.384229, -2.556783, -0.771377, 1.570796, 1.689365],accel_mss,speed_ms,0,blend_radius_m)
    |   speed_ms = 0.003
    |   movel([0.118569, -1.393867, -2.561225, -0.757297, 1.570796, 1.689365],accel_mss,speed_ms,0,blend_radius_m)
    |   speed_ms = 0.007
    |   movel([0.118728, -1.394054, -2.561089, -0.757246, 1.570796, 1.689524],accel_mss,speed_ms,0,blend_radius_m)
    |   movel([0.118593, -1.394865, -2.560501, -0.757024, 1.570796, 1.689390],accel_mss,speed_ms,0,blend_radius_m)
    |   movel([0.118424, -1.395809, -2.559814, -0.756766, 1.570796, 1.689220],accel_mss,speed_ms,0,blend_radius_m)
    |   movel([0.118206, -1.396901, -2.559018, -0.756470, 1.570796, 1.689002],accel_mss,speed_ms,0,blend_radius_m)
    |   movel([0.117896, -1.398373, -2.557942, -0.756074, 1.570796, 1.688693],accel_mss,speed_ms,0,blend_radius_m)
    |   movel([0.117699, -1.399201, -2.557336, -0.755852, 1.570796, 1.688495],accel_mss,speed_ms,0,blend_radius_m)
    |   movel([0.117545, -1.399729, -2.556948, -0.755712, 1.570796, 1.688341],accel_mss,speed_ms,0,blend_radius_m)
    |   movel([0.117303, -1.400036, -2.556723, -0.755630, 1.570796, 1.688099],accel_mss,speed_ms,0,blend_radius_m)
    |   movel([0.117055, -1.400079, -2.556692, -0.755619, 1.570796, 1.687851],accel_mss,speed_ms,0,blend_radius_m)
    |   movel([0.117023, -1.399429, -2.557168, -0.755792, 1.570796, 1.687819],accel_mss,speed_ms,0,blend_radius_m)
    |   movel([0.117111, -1.398603, -2.557774, -0.756012, 1.570796, 1.687907],accel_mss,speed_ms,0,blend_radius_m)
    |   movel([0.117305, -1.397157, -2.558831, -0.756401, 1.570796, 1.688101],accel_mss,speed_ms,0,blend_radius_m)
    |   movel([0.117464, -1.396051, -2.559637, -0.756700, 1.570796, 1.688261],accel_mss,speed_ms,0,blend_radius_m)
    |   movel([0.117616, -1.395092, -2.560336, -0.756962, 1.570796, 1.688412],accel_mss,speed_ms,0,blend_radius_m)
    |   movel([0.117758, -1.394259, -2.560940, -0.757189, 1.570796, 1.688554],accel_mss,speed_ms,0,blend_radius_m)
    |   movel([0.117985, -1.394001, -2.561128, -0.757260, 1.570796, 1.688781],accel_mss,speed_ms,0,blend_radius_m)
    |   movel([0.118280, -1.393900, -2.561201, -0.757288, 1.570796, 1.689077],accel_mss,speed_ms,0,blend_radius_m)
    |   movel([0.118569, -1.393867, -2.561225, -0.757297, 1.570796, 1.689365],accel_mss,speed_ms,0,blend_radius_m)
    |   speed_ms = 0.003
    |   movel([0.118569, -1.397123, -2.562689, -0.752577, 1.570796, 1.689365],accel_mss,speed_ms,0,blend_radius_m)
    |   speed_ms = 0.007
    |   movel([0.118728, -1.397310, -2.562553, -0.752526, 1.570796, 1.689524],accel_mss,speed_ms,0,blend_radius_m)
    |   movel([0.118593, -1.398118, -2.561963, -0.752308, 1.570796, 1.689390],accel_mss,speed_ms,0,blend_radius_m)
    |   movel([0.118424, -1.399059, -2.561275, -0.752055, 1.570796, 1.689220],accel_mss,speed_ms,0,blend_radius_m)
    |   movel([0.118206, -1.400148, -2.560477, -0.751764, 1.570796, 1.689002],accel_mss,speed_ms,0,blend_radius_m)
    |   movel([0.117896, -1.401617, -2.559399, -0.751374, 1.570796, 1.688693],accel_mss,speed_ms,0,blend_radius_m)
    |   movel([0.117699, -1.402442, -2.558791, -0.751156, 1.570796, 1.688495],accel_mss,speed_ms,0,blend_radius_m)
    |   movel([0.117545, -1.402968, -2.558403, -0.751018, 1.570796, 1.688341],accel_mss,speed_ms,0,blend_radius_m)
    |   movel([0.117303, -1.403274, -2.558177, -0.750937, 1.570796, 1.688099],accel_mss,speed_ms,0,blend_radius_m)
    |   movel([0.117055, -1.403317, -2.558145, -0.750926, 1.570796, 1.687851],accel_mss,speed_ms,0,blend_radius_m)
    |   movel([0.117023, -1.402670, -2.558623, -0.751096, 1.570796, 1.687819],accel_mss,speed_ms,0,blend_radius_m)
    |   movel([0.117111, -1.401846, -2.559230, -0.751313, 1.570796, 1.687907],accel_mss,speed_ms,0,blend_radius_m)
    |   movel([0.117305, -1.400404, -2.560290, -0.751696, 1.570796, 1.688101],accel_mss,speed_ms,0,blend_radius_m)
    |   movel([0.117464, -1.399301, -2.561098, -0.751990, 1.570796, 1.688261],accel_mss,speed_ms,0,blend_radius_m)
    |   movel([0.117616, -1.398344, -2.561798, -0.752247, 1.570796, 1.688412],accel_mss,speed_ms,0,blend_radius_m)
    |   movel([0.117758, -1.397514, -2.562404, -0.752471, 1.570796, 1.688554],accel_mss,speed_ms,0,blend_radius_m)
    |   movel([0.117985, -1.397256, -2.562592, -0.752541, 1.570796, 1.688781],accel_mss,speed_ms,0,blend_radius_m)
    |   movel([0.118280, -1.397156, -2.562665, -0.752568, 1.570796, 1.689077],accel_mss,speed_ms,0,blend_radius_m)
    |   movel([0.118569, -1.397123, -2.562689, -0.752577, 1.570796, 1.689365],accel_mss,speed_ms,0,blend_radius_m)
    |   speed_ms = 0.003
    |   movel([0.118569, -1.384229, -2.556783, -0.771377, 1.570796, 1.689365],accel_mss,speed_ms,0,blend_radius_m)
    |   speed_ms = 1.000
    |   movel([0.118569, -1.359477, -2.544576, -0.808336, 1.570796, 1.689365],accel_mss,speed_ms,0,blend_radius_m)
    |   movel([0.118605, -1.358852, -2.545007, -0.808530, 1.570796, 1.689401],accel_mss,speed_ms,0,blend_radius_m)
    |   movel([0.118605, -1.383615, -2.557221, -0.771552, 1.570796, 1.689401],accel_mss,speed_ms,0,blend_radius_m)
    |   speed_ms = 0.003
    |   movel([0.118605, -1.393258, -2.561667, -0.757465, 1.570796, 1.689401],accel_mss,speed_ms,0,blend_radius_m)
    |   speed_ms = 0.007
    |   movel([0.118234, -1.393393, -2.561569, -0.757427, 1.570796, 1.689030],accel_mss,speed_ms,0,blend_radius_m)
    |   movel([0.117908, -1.393450, -2.561527, -0.757412, 1.570796, 1.688705],accel_mss,speed_ms,0,blend_radius_m)
    |   movel([0.117689, -1.393424, -2.561546, -0.757419, 1.570796, 1.688485],accel_mss,speed_ms,0,blend_radius_m)
    |   movel([0.117549, -1.393131, -2.561759, -0.757500, 1.570796, 1.688345],accel_mss,speed_ms,0,blend_radius_m)
    |   movel([0.117522, -1.392806, -2.561994, -0.757589, 1.570796, 1.688318],accel_mss,speed_ms,0,blend_radius_m)
    |   movel([0.117346, -1.392422, -2.562271, -0.757695, 1.570796, 1.688142],accel_mss,speed_ms,0,blend_radius_m)
    |   movel([0.117088, -1.392080, -2.562518, -0.757790, 1.570796, 1.687885],accel_mss,speed_ms,0,blend_radius_m)
    |   movel([0.116802, -1.391882, -2.562661, -0.757845, 1.570796, 1.687598],accel_mss,speed_ms,0,blend_radius_m)
    |   movel([0.116439, -1.391787, -2.562731, -0.757872, 1.570796, 1.687236],accel_mss,speed_ms,0,blend_radius_m)
    |   movel([0.116040, -1.391804, -2.562718, -0.757867, 1.570796, 1.686837],accel_mss,speed_ms,0,blend_radius_m)
    |   movel([0.115619, -1.391935, -2.562624, -0.757831, 1.570796, 1.686415],accel_mss,speed_ms,0,blend_radius_m)
    |   movel([0.115183, -1.392176, -2.562449, -0.757764, 1.570796, 1.685979],accel_mss,speed_ms,0,blend_radius_m)
    |   movel([0.114712, -1.392597, -2.562145, -0.757647, 1.570796, 1.685508],accel_mss,speed_ms,0,blend_radius_m)
    |   movel([0.114471, -1.393051, -2.561816, -0.757522, 1.570796, 1.685267],accel_mss,speed_ms,0,blend_radius_m)
    |   movel([0.114501, -1.393491, -2.561498, -0.757401, 1.570796, 1.685297],accel_mss,speed_ms,0,blend_radius_m)
    |   movel([0.114790, -1.393868, -2.561224, -0.757297, 1.570796, 1.685586],accel_mss,speed_ms,0,blend_radius_m)
    |   movel([0.115093, -1.394046, -2.561095, -0.757248, 1.570796, 1.685889],accel_mss,speed_ms,0,blend_radius_m)
    |   movel([0.115465, -1.394151, -2.561019, -0.757219, 1.570796, 1.686262],accel_mss,speed_ms,0,blend_radius_m)
    |   movel([0.115948, -1.394188, -2.560992, -0.757209, 1.570796, 1.686745],accel_mss,speed_ms,0,blend_radius_m)
    |   movel([0.116596, -1.394166, -2.561008, -0.757215, 1.570796, 1.687392],accel_mss,speed_ms,0,blend_radius_m)
    |   movel([0.116840, -1.394198, -2.560985, -0.757206, 1.570796, 1.687637],accel_mss,speed_ms,0,blend_radius_m)
    |   movel([0.117037, -1.394702, -2.560619, -0.757068, 1.570796, 1.687833],accel_mss,speed_ms,0,blend_radius_m)
    |   movel([0.116741, -1.397152, -2.558834, -0.756402, 1.570796, 1.687538],accel_mss,speed_ms,0,blend_radius_m)
    |   movel([0.116430, -1.399585, -2.557054, -0.755750, 1.570796, 1.687226],accel_mss,speed_ms,0,blend_radius_m)
    |   movel([0.116267, -1.400079, -2.556692, -0.755619, 1.570796, 1.687063],accel_mss,speed_ms,0,blend_radius_m)
    |   movel([0.116071, -1.400343, -2.556497, -0.755549, 1.570796, 1.686867],accel_mss,speed_ms,0,blend_radius_m)
    |   movel([0.115806, -1.400476, -2.556399, -0.755513, 1.570796, 1.686603],accel_mss,speed_ms,0,blend_radius_m)
    |   movel([0.115532, -1.400483, -2.556394, -0.755511, 1.570796, 1.686329],accel_mss,speed_ms,0,blend_radius_m)
    |   movel([0.115371, -1.400354, -2.556490, -0.755546, 1.570796, 1.686167],accel_mss,speed_ms,0,blend_radius_m)
    |   movel([0.115306, -1.400032, -2.556726, -0.755631, 1.570796, 1.686102],accel_mss,speed_ms,0,blend_radius_m)
    |   movel([0.115324, -1.399384, -2.557202, -0.755804, 1.570796, 1.686120],accel_mss,speed_ms,0,blend_radius_m)
    |   movel([0.115335, -1.399019, -2.557469, -0.755901, 1.570796, 1.686131],accel_mss,speed_ms,0,blend_radius_m)
    |   movel([0.115328, -1.398702, -2.557701, -0.755986, 1.570796, 1.686124],accel_mss,speed_ms,0,blend_radius_m)
    |   movel([0.115303, -1.398449, -2.557887, -0.756054, 1.570796, 1.686099],accel_mss,speed_ms,0,blend_radius_m)
    |   movel([0.114943, -1.398374, -2.557941, -0.756074, 1.570796, 1.685739],accel_mss,speed_ms,0,blend_radius_m)
    |   movel([0.114662, -1.398389, -2.557930, -0.756070, 1.570796, 1.685459],accel_mss,speed_ms,0,blend_radius_m)
    |   movel([0.114357, -1.398417, -2.557910, -0.756062, 1.570796, 1.685153],accel_mss,speed_ms,0,blend_radius_m)
    |   movel([0.112719, -1.398331, -2.557973, -0.756085, 1.570796, 1.683515],accel_mss,speed_ms,0,blend_radius_m)
    |   movel([0.111315, -1.397718, -2.558421, -0.756250, 1.570796, 1.682112],accel_mss,speed_ms,0,blend_radius_m)
    |   movel([0.110329, -1.396670, -2.559187, -0.756533, 1.570796, 1.681125],accel_mss,speed_ms,0,blend_radius_m)
    |   movel([0.109898, -1.395312, -2.560175, -0.756901, 1.570796, 1.680695],accel_mss,speed_ms,0,blend_radius_m)
    |   movel([0.110008, -1.393931, -2.561179, -0.757279, 1.570796, 1.680804],accel_mss,speed_ms,0,blend_radius_m)
    |   movel([0.110561, -1.392374, -2.562306, -0.757709, 1.570796, 1.681357],accel_mss,speed_ms,0,blend_radius_m)
    |   movel([0.111504, -1.390778, -2.563459, -0.758153, 1.570796, 1.682300],accel_mss,speed_ms,0,blend_radius_m)
    |   movel([0.112755, -1.389292, -2.564528, -0.758569, 1.570796, 1.683551],accel_mss,speed_ms,0,blend_radius_m)
    |   movel([0.113901, -1.388249, -2.565277, -0.758863, 1.570796, 1.684697],accel_mss,speed_ms,0,blend_radius_m)
    |   movel([0.115113, -1.387370, -2.565906, -0.759112, 1.570796, 1.685909],accel_mss,speed_ms,0,blend_radius_m)
    |   movel([0.116414, -1.386641, -2.566428, -0.759320, 1.570796, 1.687210],accel_mss,speed_ms,0,blend_radius_m)
    |   movel([0.117832, -1.386048, -2.566851, -0.759489, 1.570796, 1.688629],accel_mss,speed_ms,0,blend_radius_m)
    |   movel([0.119207, -1.385643, -2.567141, -0.759605, 1.570796, 1.690004],accel_mss,speed_ms,0,blend_radius_m)
    |   movel([0.120533, -1.385423, -2.567298, -0.759669, 1.570796, 1.691329],accel_mss,speed_ms,0,blend_radius_m)
    |   movel([0.121802, -1.385387, -2.567323, -0.759679, 1.570796, 1.692598],accel_mss,speed_ms,0,blend_radius_m)
    |   movel([0.123004, -1.385538, -2.567216, -0.759636, 1.570796, 1.693800],accel_mss,speed_ms,0,blend_radius_m)
    |   movel([0.124432, -1.386000, -2.566886, -0.759503, 1.570796, 1.695228],accel_mss,speed_ms,0,blend_radius_m)
    |   movel([0.125530, -1.386717, -2.566374, -0.759299, 1.570796, 1.696327],accel_mss,speed_ms,0,blend_radius_m)
    |   movel([0.126289, -1.387678, -2.565686, -0.759025, 1.570796, 1.697085],accel_mss,speed_ms,0,blend_radius_m)
    |   movel([0.126698, -1.388871, -2.564830, -0.758688, 1.570796, 1.697494],accel_mss,speed_ms,0,blend_radius_m)
    |   movel([0.126745, -1.389618, -2.564293, -0.758477, 1.570796, 1.697542],accel_mss,speed_ms,0,blend_radius_m)
    |   movel([0.126649, -1.390509, -2.563652, -0.758228, 1.570796, 1.697445],accel_mss,speed_ms,0,blend_radius_m)
    |   movel([0.126428, -1.391420, -2.562996, -0.757974, 1.570796, 1.697225],accel_mss,speed_ms,0,blend_radius_m)
    |   movel([0.126106, -1.392220, -2.562417, -0.757751, 1.570796, 1.696902],accel_mss,speed_ms,0,blend_radius_m)
    |   movel([0.125118, -1.393737, -2.561319, -0.757333, 1.570796, 1.695914],accel_mss,speed_ms,0,blend_radius_m)
    |   movel([0.123745, -1.395105, -2.560326, -0.756958, 1.570796, 1.694541],accel_mss,speed_ms,0,blend_radius_m)
    |   movel([0.122153, -1.396174, -2.559548, -0.756667, 1.570796, 1.692950],accel_mss,speed_ms,0,blend_radius_m)
    |   movel([0.120525, -1.396815, -2.559081, -0.756494, 1.570796, 1.691322],accel_mss,speed_ms,0,blend_radius_m)
    |   movel([0.120253, -1.396893, -2.559024, -0.756473, 1.570796, 1.691049],accel_mss,speed_ms,0,blend_radius_m)
    |   movel([0.119842, -1.397065, -2.558898, -0.756426, 1.570796, 1.690638],accel_mss,speed_ms,0,blend_radius_m)
    |   movel([0.119569, -1.397624, -2.558489, -0.756275, 1.570796, 1.690365],accel_mss,speed_ms,0,blend_radius_m)
    |   movel([0.119430, -1.398068, -2.558166, -0.756156, 1.570796, 1.690226],accel_mss,speed_ms,0,blend_radius_m)
    |   movel([0.119286, -1.398565, -2.557802, -0.756023, 1.570796, 1.690082],accel_mss,speed_ms,0,blend_radius_m)
    |   movel([0.119073, -1.399308, -2.557257, -0.755824, 1.570796, 1.689869],accel_mss,speed_ms,0,blend_radius_m)
    |   movel([0.118949, -1.399640, -2.557014, -0.755735, 1.570796, 1.689746],accel_mss,speed_ms,0,blend_radius_m)
    |   movel([0.118677, -1.399926, -2.556804, -0.755659, 1.570796, 1.689474],accel_mss,speed_ms,0,blend_radius_m)
    |   movel([0.118374, -1.399909, -2.556816, -0.755664, 1.570796, 1.689170],accel_mss,speed_ms,0,blend_radius_m)
    |   movel([0.118256, -1.399637, -2.557016, -0.755736, 1.570796, 1.689052],accel_mss,speed_ms,0,blend_radius_m)
    |   movel([0.118338, -1.398896, -2.557559, -0.755934, 1.570796, 1.689135],accel_mss,speed_ms,0,blend_radius_m)
    |   movel([0.118759, -1.396778, -2.559108, -0.756504, 1.570796, 1.689555],accel_mss,speed_ms,0,blend_radius_m)
    |   movel([0.119135, -1.394964, -2.560428, -0.756997, 1.570796, 1.689932],accel_mss,speed_ms,0,blend_radius_m)
    |   movel([0.119322, -1.394196, -2.560986, -0.757207, 1.570796, 1.690118],accel_mss,speed_ms,0,blend_radius_m)
    |   movel([0.119471, -1.393764, -2.561299, -0.757325, 1.570796, 1.690267],accel_mss,speed_ms,0,blend_radius_m)
    |   movel([0.119650, -1.393519, -2.561478, -0.757393, 1.570796, 1.690446],accel_mss,speed_ms,0,blend_radius_m)
    |   movel([0.119894, -1.393328, -2.561616, -0.757445, 1.570796, 1.690690],accel_mss,speed_ms,0,blend_radius_m)
    |   movel([0.120184, -1.393181, -2.561722, -0.757486, 1.570796, 1.690980],accel_mss,speed_ms,0,blend_radius_m)
    |   movel([0.120541, -1.392912, -2.561917, -0.757560, 1.570796, 1.691338],accel_mss,speed_ms,0,blend_radius_m)
    |   movel([0.121356, -1.391952, -2.562611, -0.757826, 1.570796, 1.692152],accel_mss,speed_ms,0,blend_radius_m)
    |   movel([0.121511, -1.391218, -2.563141, -0.758030, 1.570796, 1.692307],accel_mss,speed_ms,0,blend_radius_m)
    |   movel([0.121159, -1.390779, -2.563458, -0.758152, 1.570796, 1.691955],accel_mss,speed_ms,0,blend_radius_m)
    |   movel([0.120423, -1.390764, -2.563469, -0.758157, 1.570796, 1.691219],accel_mss,speed_ms,0,blend_radius_m)
    |   movel([0.119974, -1.390949, -2.563335, -0.758105, 1.570796, 1.690770],accel_mss,speed_ms,0,blend_radius_m)
    |   movel([0.119626, -1.391236, -2.563128, -0.758025, 1.570796, 1.690422],accel_mss,speed_ms,0,blend_radius_m)
    |   movel([0.119362, -1.391651, -2.562829, -0.757909, 1.570796, 1.690158],accel_mss,speed_ms,0,blend_radius_m)
    |   movel([0.119164, -1.392229, -2.562411, -0.757749, 1.570796, 1.689960],accel_mss,speed_ms,0,blend_radius_m)
    |   movel([0.118997, -1.392786, -2.562008, -0.757595, 1.570796, 1.689793],accel_mss,speed_ms,0,blend_radius_m)
    |   movel([0.118834, -1.393077, -2.561797, -0.757514, 1.570796, 1.689630],accel_mss,speed_ms,0,blend_radius_m)
    |   movel([0.118605, -1.393258, -2.561667, -0.757465, 1.570796, 1.689401],accel_mss,speed_ms,0,blend_radius_m)
    |   speed_ms = 0.003
    |   movel([0.118605, -1.396515, -2.563132, -0.752742, 1.570796, 1.689401],accel_mss,speed_ms,0,blend_radius_m)
    |   speed_ms = 0.007
    |   movel([0.118234, -1.396650, -2.563034, -0.752705, 1.570796, 1.689030],accel_mss,speed_ms,0,blend_radius_m)
    |   movel([0.117908, -1.396707, -2.562992, -0.752690, 1.570796, 1.688705],accel_mss,speed_ms,0,blend_radius_m)
    |   movel([0.117689, -1.396681, -2.563011, -0.752697, 1.570796, 1.688485],accel_mss,speed_ms,0,blend_radius_m)
    |   movel([0.117549, -1.396389, -2.563224, -0.752776, 1.570796, 1.688345],accel_mss,speed_ms,0,blend_radius_m)
    |   movel([0.117522, -1.396065, -2.563460, -0.752865, 1.570796, 1.688318],accel_mss,speed_ms,0,blend_radius_m)
    |   movel([0.117346, -1.395682, -2.563738, -0.752969, 1.570796, 1.688142],accel_mss,speed_ms,0,blend_radius_m)
    |   movel([0.117088, -1.395341, -2.563985, -0.753062, 1.570796, 1.687885],accel_mss,speed_ms,0,blend_radius_m)
    |   movel([0.116802, -1.395144, -2.564129, -0.753116, 1.570796, 1.687598],accel_mss,speed_ms,0,blend_radius_m)
    |   movel([0.116439, -1.395048, -2.564198, -0.753143, 1.570796, 1.687236],accel_mss,speed_ms,0,blend_radius_m)
    |   movel([0.116040, -1.395066, -2.564185, -0.753138, 1.570796, 1.686837],accel_mss,speed_ms,0,blend_radius_m)
    |   movel([0.115619, -1.395196, -2.564091, -0.753102, 1.570796, 1.686415],accel_mss,speed_ms,0,blend_radius_m)
    |   movel([0.115183, -1.395437, -2.563916, -0.753036, 1.570796, 1.685979],accel_mss,speed_ms,0,blend_radius_m)
    |   movel([0.114712, -1.395856, -2.563611, -0.752922, 1.570796, 1.685508],accel_mss,speed_ms,0,blend_radius_m)
    |   movel([0.114471, -1.396309, -2.563281, -0.752798, 1.570796, 1.685267],accel_mss,speed_ms,0,blend_radius_m)
    |   movel([0.114501, -1.396748, -2.562962, -0.752679, 1.570796, 1.685297],accel_mss,speed_ms,0,blend_radius_m)
    |   movel([0.114790, -1.397124, -2.562688, -0.752577, 1.570796, 1.685586],accel_mss,speed_ms,0,blend_radius_m)
    |   movel([0.115093, -1.397302, -2.562559, -0.752529, 1.570796, 1.685889],accel_mss,speed_ms,0,blend_radius_m)
    |   movel([0.115465, -1.397406, -2.562482, -0.752500, 1.570796, 1.686262],accel_mss,speed_ms,0,blend_radius_m)
    |   movel([0.115948, -1.397443, -2.562455, -0.752490, 1.570796, 1.686745],accel_mss,speed_ms,0,blend_radius_m)
    |   movel([0.116596, -1.397422, -2.562471, -0.752496, 1.570796, 1.687392],accel_mss,speed_ms,0,blend_radius_m)
    |   movel([0.116840, -1.397453, -2.562448, -0.752488, 1.570796, 1.687637],accel_mss,speed_ms,0,blend_radius_m)
    |   movel([0.117037, -1.397956, -2.562081, -0.752352, 1.570796, 1.687833],accel_mss,speed_ms,0,blend_radius_m)
    |   movel([0.116741, -1.400399, -2.560293, -0.751697, 1.570796, 1.687538],accel_mss,speed_ms,0,blend_radius_m)
    |   movel([0.116430, -1.402825, -2.558508, -0.751055, 1.570796, 1.687226],accel_mss,speed_ms,0,blend_radius_m)
    |   movel([0.116267, -1.403317, -2.558146, -0.750926, 1.570796, 1.687063],accel_mss,speed_ms,0,blend_radius_m)
    |   movel([0.116071, -1.403581, -2.557951, -0.750857, 1.570796, 1.686867],accel_mss,speed_ms,0,blend_radius_m)
    |   movel([0.115806, -1.403714, -2.557853, -0.750822, 1.570796, 1.686603],accel_mss,speed_ms,0,blend_radius_m)
    |   movel([0.115532, -1.403721, -2.557848, -0.750821, 1.570796, 1.686329],accel_mss,speed_ms,0,blend_radius_m)
    |   movel([0.115371, -1.403591, -2.557943, -0.750854, 1.570796, 1.686167],accel_mss,speed_ms,0,blend_radius_m)
    |   movel([0.115306, -1.403270, -2.558180, -0.750938, 1.570796, 1.686102],accel_mss,speed_ms,0,blend_radius_m)
    |   movel([0.115324, -1.402624, -2.558657, -0.751108, 1.570796, 1.686120],accel_mss,speed_ms,0,blend_radius_m)
    |   movel([0.115335, -1.402261, -2.558925, -0.751204, 1.570796, 1.686131],accel_mss,speed_ms,0,blend_radius_m)
    |   movel([0.115328, -1.401944, -2.559157, -0.751287, 1.570796, 1.686124],accel_mss,speed_ms,0,blend_radius_m)
    |   movel([0.115303, -1.401692, -2.559343, -0.751354, 1.570796, 1.686099],accel_mss,speed_ms,0,blend_radius_m)
    |   movel([0.114943, -1.401617, -2.559398, -0.751374, 1.570796, 1.685739],accel_mss,speed_ms,0,blend_radius_m)
    |   movel([0.114662, -1.401633, -2.559387, -0.751370, 1.570796, 1.685459],accel_mss,speed_ms,0,blend_radius_m)
    |   movel([0.114357, -1.401660, -2.559366, -0.751362, 1.570796, 1.685153],accel_mss,speed_ms,0,blend_radius_m)
    |   movel([0.112719, -1.401575, -2.559429, -0.751385, 1.570796, 1.683515],accel_mss,speed_ms,0,blend_radius_m)
    |   movel([0.111315, -1.400963, -2.559879, -0.751547, 1.570796, 1.682112],accel_mss,speed_ms,0,blend_radius_m)
    |   movel([0.110329, -1.399918, -2.560646, -0.751825, 1.570796, 1.681125],accel_mss,speed_ms,0,blend_radius_m)
    |   movel([0.109898, -1.398564, -2.561637, -0.752188, 1.570796, 1.680695],accel_mss,speed_ms,0,blend_radius_m)
    |   movel([0.110008, -1.397187, -2.562642, -0.752560, 1.570796, 1.680804],accel_mss,speed_ms,0,blend_radius_m)
    |   movel([0.110561, -1.395634, -2.563773, -0.752982, 1.570796, 1.681357],accel_mss,speed_ms,0,blend_radius_m)
    |   movel([0.111504, -1.394042, -2.564928, -0.753419, 1.570796, 1.682300],accel_mss,speed_ms,0,blend_radius_m)
    |   movel([0.112755, -1.392561, -2.565999, -0.753829, 1.570796, 1.683551],accel_mss,speed_ms,0,blend_radius_m)
    |   movel([0.113901, -1.391520, -2.566750, -0.754119, 1.570796, 1.684697],accel_mss,speed_ms,0,blend_radius_m)
    |   movel([0.115113, -1.390644, -2.567381, -0.754364, 1.570796, 1.685909],accel_mss,speed_ms,0,blend_radius_m)
    |   movel([0.116414, -1.389917, -2.567904, -0.754568, 1.570796, 1.687210],accel_mss,speed_ms,0,blend_radius_m)
    |   movel([0.117832, -1.389326, -2.568328, -0.754735, 1.570796, 1.688629],accel_mss,speed_ms,0,blend_radius_m)
    |   movel([0.119207, -1.388922, -2.568618, -0.754849, 1.570796, 1.690004],accel_mss,speed_ms,0,blend_radius_m)
    |   movel([0.120533, -1.388702, -2.568775, -0.754912, 1.570796, 1.691329],accel_mss,speed_ms,0,blend_radius_m)
    |   movel([0.121802, -1.388667, -2.568801, -0.754922, 1.570796, 1.692598],accel_mss,speed_ms,0,blend_radius_m)
    |   movel([0.123004, -1.388816, -2.568693, -0.754879, 1.570796, 1.693800],accel_mss,speed_ms,0,blend_radius_m)
    |   movel([0.124432, -1.389277, -2.568363, -0.754749, 1.570796, 1.695228],accel_mss,speed_ms,0,blend_radius_m)
    |   movel([0.125530, -1.389992, -2.567850, -0.754547, 1.570796, 1.696327],accel_mss,speed_ms,0,blend_radius_m)
    |   movel([0.126289, -1.390951, -2.567160, -0.754278, 1.570796, 1.697085],accel_mss,speed_ms,0,blend_radius_m)
    |   movel([0.126698, -1.392141, -2.566302, -0.753946, 1.570796, 1.697494],accel_mss,speed_ms,0,blend_radius_m)
    |   movel([0.126745, -1.392886, -2.565764, -0.753739, 1.570796, 1.697542],accel_mss,speed_ms,0,blend_radius_m)
    |   movel([0.126649, -1.393774, -2.565122, -0.753493, 1.570796, 1.697445],accel_mss,speed_ms,0,blend_radius_m)
    |   movel([0.126428, -1.394682, -2.564464, -0.753243, 1.570796, 1.697225],accel_mss,speed_ms,0,blend_radius_m)
    |   movel([0.126106, -1.395481, -2.563884, -0.753024, 1.570796, 1.696902],accel_mss,speed_ms,0,blend_radius_m)
    |   movel([0.125118, -1.396993, -2.562784, -0.752612, 1.570796, 1.695914],accel_mss,speed_ms,0,blend_radius_m)
    |   movel([0.123745, -1.398357, -2.561788, -0.752244, 1.570796, 1.694541],accel_mss,speed_ms,0,blend_radius_m)
    |   movel([0.122153, -1.399423, -2.561008, -0.751957, 1.570796, 1.692950],accel_mss,speed_ms,0,blend_radius_m)
    |   movel([0.120525, -1.400063, -2.560540, -0.751787, 1.570796, 1.691322],accel_mss,speed_ms,0,blend_radius_m)
    |   movel([0.120253, -1.400140, -2.560483, -0.751766, 1.570796, 1.691049],accel_mss,speed_ms,0,blend_radius_m)
    |   movel([0.119842, -1.400312, -2.560357, -0.751720, 1.570796, 1.690638],accel_mss,speed_ms,0,blend_radius_m)
    |   movel([0.119569, -1.400870, -2.559947, -0.751572, 1.570796, 1.690365],accel_mss,speed_ms,0,blend_radius_m)
    |   movel([0.119430, -1.401312, -2.559623, -0.751455, 1.570796, 1.690226],accel_mss,speed_ms,0,blend_radius_m)
    |   movel([0.119286, -1.401808, -2.559258, -0.751323, 1.570796, 1.690082],accel_mss,speed_ms,0,blend_radius_m)
    |   movel([0.119073, -1.402549, -2.558712, -0.751128, 1.570796, 1.689869],accel_mss,speed_ms,0,blend_radius_m)
    |   movel([0.118949, -1.402880, -2.558468, -0.751041, 1.570796, 1.689746],accel_mss,speed_ms,0,blend_radius_m)
    |   movel([0.118677, -1.403165, -2.558258, -0.750966, 1.570796, 1.689474],accel_mss,speed_ms,0,blend_radius_m)
    |   movel([0.118374, -1.403148, -2.558270, -0.750970, 1.570796, 1.689170],accel_mss,speed_ms,0,blend_radius_m)
    |   movel([0.118256, -1.402877, -2.558470, -0.751042, 1.570796, 1.689052],accel_mss,speed_ms,0,blend_radius_m)
    |   movel([0.118338, -1.402138, -2.559015, -0.751236, 1.570796, 1.689135],accel_mss,speed_ms,0,blend_radius_m)
    |   movel([0.118759, -1.400026, -2.560567, -0.751796, 1.570796, 1.689555],accel_mss,speed_ms,0,blend_radius_m)
    |   movel([0.119135, -1.398217, -2.561891, -0.752281, 1.570796, 1.689932],accel_mss,speed_ms,0,blend_radius_m)
    |   movel([0.119322, -1.397451, -2.562450, -0.752488, 1.570796, 1.690118],accel_mss,speed_ms,0,blend_radius_m)
    |   movel([0.119471, -1.397021, -2.562764, -0.752605, 1.570796, 1.690267],accel_mss,speed_ms,0,blend_radius_m)
    |   movel([0.119650, -1.396776, -2.562942, -0.752671, 1.570796, 1.690446],accel_mss,speed_ms,0,blend_radius_m)
    |   movel([0.119894, -1.396586, -2.563080, -0.752723, 1.570796, 1.690690],accel_mss,speed_ms,0,blend_radius_m)
    |   movel([0.120184, -1.396439, -2.563187, -0.752763, 1.570796, 1.690980],accel_mss,speed_ms,0,blend_radius_m)
    |   movel([0.120541, -1.396171, -2.563382, -0.752836, 1.570796, 1.691338],accel_mss,speed_ms,0,blend_radius_m)
    |   movel([0.121356, -1.395214, -2.564078, -0.753097, 1.570796, 1.692152],accel_mss,speed_ms,0,blend_radius_m)
    |   movel([0.121511, -1.394481, -2.564609, -0.753298, 1.570796, 1.692307],accel_mss,speed_ms,0,blend_radius_m)
    |   movel([0.121159, -1.394043, -2.564927, -0.753419, 1.570796, 1.691955],accel_mss,speed_ms,0,blend_radius_m)
    |   movel([0.120423, -1.394028, -2.564938, -0.753423, 1.570796, 1.691219],accel_mss,speed_ms,0,blend_radius_m)
    |   movel([0.119974, -1.394213, -2.564804, -0.753372, 1.570796, 1.690770],accel_mss,speed_ms,0,blend_radius_m)
    |   movel([0.119626, -1.394499, -2.564597, -0.753293, 1.570796, 1.690422],accel_mss,speed_ms,0,blend_radius_m)
    |   movel([0.119362, -1.394913, -2.564296, -0.753180, 1.570796, 1.690158],accel_mss,speed_ms,0,blend_radius_m)
    |   movel([0.119164, -1.395489, -2.563878, -0.753022, 1.570796, 1.689960],accel_mss,speed_ms,0,blend_radius_m)
    |   movel([0.118997, -1.396045, -2.563474, -0.752870, 1.570796, 1.689793],accel_mss,speed_ms,0,blend_radius_m)
    |   movel([0.118834, -1.396335, -2.563263, -0.752791, 1.570796, 1.689630],accel_mss,speed_ms,0,blend_radius_m)
    |   movel([0.118605, -1.396515, -2.563132, -0.752742, 1.570796, 1.689401],accel_mss,speed_ms,0,blend_radius_m)
    |   speed_ms = 0.003
    |   movel([0.118605, -1.383615, -2.557221, -0.771552, 1.570796, 1.689401],accel_mss,speed_ms,0,blend_radius_m)
    |   speed_ms = 1.000
    |   movel([0.118605, -1.358852, -2.545007, -0.808530, 1.570796, 1.689401],accel_mss,speed_ms,0,blend_radius_m)
    |   movel([0.116923, -1.366587, -2.539643, -0.806159, 1.570796, 1.687720],accel_mss,speed_ms,0,blend_radius_m)
    |   movel([0.116923, -1.391208, -2.551760, -0.769421, 1.570796, 1.687720],accel_mss,speed_ms,0,blend_radius_m)
    |   speed_ms = 0.003
    |   movel([0.116923, -1.400790, -2.556169, -0.755430, 1.570796, 1.687720],accel_mss,speed_ms,0,blend_radius_m)
    |   speed_ms = 0.007
    |   movel([0.118450, -1.400541, -2.556352, -0.755496, 1.570796, 1.689246],accel_mss,speed_ms,0,blend_radius_m)
    |   movel([0.119164, -1.400486, -2.556392, -0.755511, 1.570796, 1.689961],accel_mss,speed_ms,0,blend_radius_m)
    |   movel([0.119522, -1.400571, -2.556330, -0.755488, 1.570796, 1.690318],accel_mss,speed_ms,0,blend_radius_m)
    |   movel([0.119673, -1.400804, -2.556159, -0.755426, 1.570796, 1.690469],accel_mss,speed_ms,0,blend_radius_m)
    |   movel([0.119491, -1.401099, -2.555942, -0.755349, 1.570796, 1.690287],accel_mss,speed_ms,0,blend_radius_m)
    |   movel([0.119212, -1.401506, -2.555642, -0.755241, 1.570796, 1.690008],accel_mss,speed_ms,0,blend_radius_m)
    |   movel([0.119126, -1.401821, -2.555410, -0.755158, 1.570796, 1.689922],accel_mss,speed_ms,0,blend_radius_m)
    |   movel([0.119166, -1.402025, -2.555260, -0.755105, 1.570796, 1.689962],accel_mss,speed_ms,0,blend_radius_m)
    |   movel([0.119206, -1.402226, -2.555111, -0.755052, 1.570796, 1.690002],accel_mss,speed_ms,0,blend_radius_m)
    |   movel([0.119129, -1.402510, -2.554902, -0.754977, 1.570796, 1.689926],accel_mss,speed_ms,0,blend_radius_m)
    |   movel([0.118545, -1.403144, -2.554433, -0.754811, 1.570796, 1.689342],accel_mss,speed_ms,0,blend_radius_m)
    |   movel([0.118026, -1.403479, -2.554186, -0.754724, 1.570796, 1.688823],accel_mss,speed_ms,0,blend_radius_m)
    |   movel([0.117329, -1.403764, -2.553976, -0.754650, 1.570796, 1.688126],accel_mss,speed_ms,0,blend_radius_m)
    |   movel([0.116307, -1.404052, -2.553762, -0.754575, 1.570796, 1.687103],accel_mss,speed_ms,0,blend_radius_m)
    |   movel([0.115098, -1.404316, -2.553567, -0.754506, 1.570796, 1.685894],accel_mss,speed_ms,0,blend_radius_m)
    |   movel([0.114445, -1.404324, -2.553560, -0.754504, 1.570796, 1.685242],accel_mss,speed_ms,0,blend_radius_m)
    |   movel([0.114245, -1.404102, -2.553725, -0.754562, 1.570796, 1.685042],accel_mss,speed_ms,0,blend_radius_m)
    |   movel([0.114389, -1.403691, -2.554029, -0.754669, 1.570796, 1.685185],accel_mss,speed_ms,0,blend_radius_m)
    |   movel([0.114487, -1.403461, -2.554199, -0.754729, 1.570796, 1.685284],accel_mss,speed_ms,0,blend_radius_m)
    |   movel([0.114325, -1.403271, -2.554340, -0.754778, 1.570796, 1.685121],accel_mss,speed_ms,0,blend_radius_m)
    |   movel([0.114088, -1.403092, -2.554472, -0.754825, 1.570796, 1.684885],accel_mss,speed_ms,0,blend_radius_m)
    |   movel([0.114422, -1.402771, -2.554709, -0.754909, 1.570796, 1.685218],accel_mss,speed_ms,0,blend_radius_m)
    |   movel([0.114756, -1.402449, -2.554947, -0.754993, 1.570796, 1.685552],accel_mss,speed_ms,0,blend_radius_m)
    |   movel([0.114495, -1.402217, -2.555118, -0.755054, 1.570796, 1.685292],accel_mss,speed_ms,0,blend_radius_m)
    |   movel([0.114323, -1.402013, -2.555268, -0.755108, 1.570796, 1.685119],accel_mss,speed_ms,0,blend_radius_m)
    |   movel([0.114274, -1.401816, -2.555414, -0.755159, 1.570796, 1.685070],accel_mss,speed_ms,0,blend_radius_m)
    |   movel([0.114523, -1.401391, -2.555726, -0.755271, 1.570796, 1.685319],accel_mss,speed_ms,0,blend_radius_m)
    |   movel([0.115063, -1.401146, -2.555907, -0.755336, 1.570796, 1.685859],accel_mss,speed_ms,0,blend_radius_m)
    |   movel([0.115634, -1.401022, -2.555998, -0.755369, 1.570796, 1.686431],accel_mss,speed_ms,0,blend_radius_m)
    |   movel([0.116923, -1.400790, -2.556169, -0.755430, 1.570796, 1.687720],accel_mss,speed_ms,0,blend_radius_m)
    |   speed_ms = 0.003
    |   movel([0.116923, -1.404026, -2.557622, -0.750741, 1.570796, 1.687720],accel_mss,speed_ms,0,blend_radius_m)
    |   speed_ms = 0.007
    |   movel([0.118450, -1.403778, -2.557805, -0.750806, 1.570796, 1.689246],accel_mss,speed_ms,0,blend_radius_m)
    |   movel([0.119164, -1.403723, -2.557846, -0.750820, 1.570796, 1.689961],accel_mss,speed_ms,0,blend_radius_m)
    |   movel([0.119522, -1.403808, -2.557783, -0.750798, 1.570796, 1.690318],accel_mss,speed_ms,0,blend_radius_m)
    |   movel([0.119673, -1.404040, -2.557611, -0.750737, 1.570796, 1.690469],accel_mss,speed_ms,0,blend_radius_m)
    |   movel([0.119491, -1.404334, -2.557394, -0.750660, 1.570796, 1.690287],accel_mss,speed_ms,0,blend_radius_m)
    |   movel([0.119212, -1.404740, -2.557094, -0.750555, 1.570796, 1.690008],accel_mss,speed_ms,0,blend_radius_m)
    |   movel([0.119126, -1.405055, -2.556861, -0.750473, 1.570796, 1.689922],accel_mss,speed_ms,0,blend_radius_m)
    |   movel([0.119166, -1.405258, -2.556711, -0.750421, 1.570796, 1.689962],accel_mss,speed_ms,0,blend_radius_m)
    |   movel([0.119206, -1.405459, -2.556562, -0.750369, 1.570796, 1.690002],accel_mss,speed_ms,0,blend_radius_m)
    |   movel([0.119129, -1.405742, -2.556352, -0.750295, 1.570796, 1.689926],accel_mss,speed_ms,0,blend_radius_m)
    |   movel([0.118545, -1.406374, -2.555882, -0.750132, 1.570796, 1.689342],accel_mss,speed_ms,0,blend_radius_m)
    |   movel([0.118026, -1.406708, -2.555634, -0.750046, 1.570796, 1.688823],accel_mss,speed_ms,0,blend_radius_m)
    |   movel([0.117329, -1.406992, -2.555424, -0.749974, 1.570796, 1.688126],accel_mss,speed_ms,0,blend_radius_m)
    |   movel([0.116307, -1.407280, -2.555210, -0.749900, 1.570796, 1.687103],accel_mss,speed_ms,0,blend_radius_m)
    |   movel([0.115098, -1.407542, -2.555014, -0.749833, 1.570796, 1.685894],accel_mss,speed_ms,0,blend_radius_m)
    |   movel([0.114445, -1.407551, -2.555008, -0.749830, 1.570796, 1.685242],accel_mss,speed_ms,0,blend_radius_m)
    |   movel([0.114245, -1.407329, -2.555173, -0.749887, 1.570796, 1.685042],accel_mss,speed_ms,0,blend_radius_m)
    |   movel([0.114389, -1.406920, -2.555477, -0.749992, 1.570796, 1.685185],accel_mss,speed_ms,0,blend_radius_m)
    |   movel([0.114487, -1.406690, -2.555648, -0.750051, 1.570796, 1.685284],accel_mss,speed_ms,0,blend_radius_m)
    |   movel([0.114325, -1.406501, -2.555788, -0.750100, 1.570796, 1.685121],accel_mss,speed_ms,0,blend_radius_m)
    |   movel([0.114088, -1.406322, -2.555921, -0.750146, 1.570796, 1.684885],accel_mss,speed_ms,0,blend_radius_m)
    |   movel([0.114422, -1.406002, -2.556159, -0.750228, 1.570796, 1.685218],accel_mss,speed_ms,0,blend_radius_m)
    |   movel([0.114756, -1.405681, -2.556397, -0.750311, 1.570796, 1.685552],accel_mss,speed_ms,0,blend_radius_m)
    |   movel([0.114495, -1.405449, -2.556569, -0.750371, 1.570796, 1.685292],accel_mss,speed_ms,0,blend_radius_m)
    |   movel([0.114323, -1.405246, -2.556719, -0.750424, 1.570796, 1.685119],accel_mss,speed_ms,0,blend_radius_m)
    |   movel([0.114274, -1.405050, -2.556865, -0.750475, 1.570796, 1.685070],accel_mss,speed_ms,0,blend_radius_m)
    |   movel([0.114523, -1.404626, -2.557178, -0.750585, 1.570796, 1.685319],accel_mss,speed_ms,0,blend_radius_m)
    |   movel([0.115063, -1.404382, -2.557359, -0.750648, 1.570796, 1.685859],accel_mss,speed_ms,0,blend_radius_m)
    |   movel([0.115634, -1.404258, -2.557451, -0.750680, 1.570796, 1.686431],accel_mss,speed_ms,0,blend_radius_m)
    |   movel([0.116923, -1.404026, -2.557622, -0.750741, 1.570796, 1.687720],accel_mss,speed_ms,0,blend_radius_m)
    |   speed_ms = 0.003
    |   movel([0.116923, -1.391208, -2.551760, -0.769421, 1.570796, 1.687720],accel_mss,speed_ms,0,blend_radius_m)
    |   speed_ms = 1.000
    |   movel([0.116923, -1.366587, -2.539643, -0.806159, 1.570796, 1.687720],accel_mss,speed_ms,0,blend_radius_m)
    |   movel([0.116275, -1.370444, -2.536938, -0.805007, 1.570796, 1.687072],accel_mss,speed_ms,0,blend_radius_m)
    |   movel([0.116275, -1.394993, -2.549006, -0.768389, 1.570796, 1.687072],accel_mss,speed_ms,0,blend_radius_m)
    |   speed_ms = 0.003
    |   movel([0.116275, -1.404545, -2.553397, -0.754447, 1.570796, 1.687072],accel_mss,speed_ms,0,blend_radius_m)
    |   speed_ms = 0.007
    |   movel([0.116705, -1.404434, -2.553479, -0.754476, 1.570796, 1.687501],accel_mss,speed_ms,0,blend_radius_m)
    |   movel([0.117062, -1.404455, -2.553464, -0.754470, 1.570796, 1.687859],accel_mss,speed_ms,0,blend_radius_m)
    |   movel([0.117167, -1.404617, -2.553344, -0.754428, 1.570796, 1.687963],accel_mss,speed_ms,0,blend_radius_m)
    |   movel([0.116942, -1.404907, -2.553129, -0.754353, 1.570796, 1.687739],accel_mss,speed_ms,0,blend_radius_m)
    |   movel([0.116708, -1.405086, -2.552996, -0.754307, 1.570796, 1.687504],accel_mss,speed_ms,0,blend_radius_m)
    |   movel([0.116444, -1.405186, -2.552922, -0.754281, 1.570796, 1.687240],accel_mss,speed_ms,0,blend_radius_m)
    |   movel([0.116190, -1.405195, -2.552915, -0.754279, 1.570796, 1.686986],accel_mss,speed_ms,0,blend_radius_m)
    |   movel([0.115991, -1.405108, -2.552980, -0.754301, 1.570796, 1.686788],accel_mss,speed_ms,0,blend_radius_m)
    |   movel([0.115873, -1.404946, -2.553100, -0.754343, 1.570796, 1.686669],accel_mss,speed_ms,0,blend_radius_m)
    |   movel([0.116275, -1.404545, -2.553397, -0.754447, 1.570796, 1.687072],accel_mss,speed_ms,0,blend_radius_m)
    |   speed_ms = 0.003
    |   movel([0.116275, -1.407771, -2.554844, -0.749774, 1.570796, 1.687072],accel_mss,speed_ms,0,blend_radius_m)
    |   speed_ms = 0.007
    |   movel([0.116705, -1.407660, -2.554926, -0.749802, 1.570796, 1.687501],accel_mss,speed_ms,0,blend_radius_m)
    |   movel([0.117062, -1.407681, -2.554911, -0.749797, 1.570796, 1.687859],accel_mss,speed_ms,0,blend_radius_m)
    |   movel([0.117167, -1.407843, -2.554790, -0.749756, 1.570796, 1.687963],accel_mss,speed_ms,0,blend_radius_m)
    |   movel([0.116942, -1.408132, -2.554575, -0.749682, 1.570796, 1.687739],accel_mss,speed_ms,0,blend_radius_m)
    |   movel([0.116708, -1.408311, -2.554442, -0.749637, 1.570796, 1.687504],accel_mss,speed_ms,0,blend_radius_m)
    |   movel([0.116444, -1.408410, -2.554368, -0.749611, 1.570796, 1.687240],accel_mss,speed_ms,0,blend_radius_m)
    |   movel([0.116190, -1.408420, -2.554361, -0.749609, 1.570796, 1.686986],accel_mss,speed_ms,0,blend_radius_m)
    |   movel([0.115991, -1.408333, -2.554425, -0.749631, 1.570796, 1.686788],accel_mss,speed_ms,0,blend_radius_m)
    |   movel([0.115873, -1.408171, -2.554546, -0.749672, 1.570796, 1.686669],accel_mss,speed_ms,0,blend_radius_m)
    |   movel([0.116275, -1.407771, -2.554844, -0.749774, 1.570796, 1.687072],accel_mss,speed_ms,0,blend_radius_m)
    |   speed_ms = 0.003
    |   movel([0.116275, -1.394993, -2.549006, -0.768389, 1.570796, 1.687072],accel_mss,speed_ms,0,blend_radius_m)
    |   speed_ms = 1.000
    |   movel([0.116275, -1.370444, -2.536938, -0.805007, 1.570796, 1.687072],accel_mss,speed_ms,0,blend_radius_m)
    |   movel([0.071617, -1.356963, -2.546304, -0.809122, 1.570796, 1.642413],accel_mss,speed_ms,0,blend_radius_m)
    |   movel([0.071617, -1.381761, -2.558542, -0.772086, 1.570796, 1.642413],accel_mss,speed_ms,0,blend_radius_m)
    |   speed_ms = 0.003
    |   movel([0.071617, -1.391418, -2.562997, -0.757974, 1.570796, 1.642413],accel_mss,speed_ms,0,blend_radius_m)
    |   speed_ms = 0.007
    |   movel([0.069577, -1.391884, -2.562661, -0.757845, 1.570796, 1.640373],accel_mss,speed_ms,0,blend_radius_m)
    |   movel([0.068922, -1.391989, -2.562584, -0.757815, 1.570796, 1.639718],accel_mss,speed_ms,0,blend_radius_m)
    |   movel([0.068598, -1.391994, -2.562581, -0.757814, 1.570796, 1.639395],accel_mss,speed_ms,0,blend_radius_m)
    |   movel([0.068461, -1.391838, -2.562694, -0.757857, 1.570796, 1.639258],accel_mss,speed_ms,0,blend_radius_m)
    |   movel([0.068638, -1.391563, -2.562892, -0.757934, 1.570796, 1.639434],accel_mss,speed_ms,0,blend_radius_m)
    |   movel([0.069122, -1.391247, -2.563120, -0.758022, 1.570796, 1.639918],accel_mss,speed_ms,0,blend_radius_m)
    |   movel([0.070213, -1.390930, -2.563349, -0.758110, 1.570796, 1.641009],accel_mss,speed_ms,0,blend_radius_m)
    |   movel([0.071290, -1.390711, -2.563507, -0.758171, 1.570796, 1.642087],accel_mss,speed_ms,0,blend_radius_m)
    |   movel([0.071672, -1.390815, -2.563432, -0.758142, 1.570796, 1.642469],accel_mss,speed_ms,0,blend_radius_m)
    |   movel([0.071727, -1.391083, -2.563239, -0.758068, 1.570796, 1.642523],accel_mss,speed_ms,0,blend_radius_m)
    |   movel([0.071675, -1.391329, -2.563061, -0.757999, 1.570796, 1.642471],accel_mss,speed_ms,0,blend_radius_m)
    |   speed_ms = 0.003
    |   movel([0.071617, -1.394681, -2.564465, -0.753243, 1.570796, 1.642413],accel_mss,speed_ms,0,blend_radius_m)
    |   speed_ms = 0.007
    |   movel([0.069577, -1.395145, -2.564128, -0.753116, 1.570796, 1.640373],accel_mss,speed_ms,0,blend_radius_m)
    |   movel([0.068922, -1.395251, -2.564051, -0.753087, 1.570796, 1.639718],accel_mss,speed_ms,0,blend_radius_m)
    |   movel([0.068598, -1.395255, -2.564048, -0.753086, 1.570796, 1.639395],accel_mss,speed_ms,0,blend_radius_m)
    |   movel([0.068461, -1.395099, -2.564161, -0.753129, 1.570796, 1.639258],accel_mss,speed_ms,0,blend_radius_m)
    |   movel([0.068638, -1.394825, -2.564360, -0.753204, 1.570796, 1.639434],accel_mss,speed_ms,0,blend_radius_m)
    |   movel([0.069122, -1.394510, -2.564589, -0.753290, 1.570796, 1.639918],accel_mss,speed_ms,0,blend_radius_m)
    |   movel([0.070213, -1.394194, -2.564818, -0.753377, 1.570796, 1.641009],accel_mss,speed_ms,0,blend_radius_m)
    |   movel([0.071290, -1.393975, -2.564976, -0.753438, 1.570796, 1.642087],accel_mss,speed_ms,0,blend_radius_m)
    |   movel([0.071672, -1.394079, -2.564901, -0.753409, 1.570796, 1.642469],accel_mss,speed_ms,0,blend_radius_m)
    |   movel([0.071727, -1.394346, -2.564707, -0.753335, 1.570796, 1.642523],accel_mss,speed_ms,0,blend_radius_m)
    |   movel([0.071675, -1.394592, -2.564529, -0.753268, 1.570796, 1.642471],accel_mss,speed_ms,0,blend_radius_m)
    |   speed_ms = 0.003
    |   movel([0.071617, -1.381761, -2.558542, -0.772086, 1.570796, 1.642413],accel_mss,speed_ms,0,blend_radius_m)
    |   speed_ms = 1.000
    |   movel([0.071617, -1.356963, -2.546304, -0.809122, 1.570796, 1.642413],accel_mss,speed_ms,0,blend_radius_m)
    |   movel([0.071390, -1.355193, -2.547515, -0.809680, 1.570796, 1.642186],accel_mss,speed_ms,0,blend_radius_m)
    |   movel([0.071390, -1.380023, -2.559776, -0.772590, 1.570796, 1.642186],accel_mss,speed_ms,0,blend_radius_m)
    |   speed_ms = 0.003
    |   movel([0.071390, -1.389694, -2.564239, -0.758456, 1.570796, 1.642186],accel_mss,speed_ms,0,blend_radius_m)
    |   speed_ms = 0.007
    |   movel([0.071125, -1.389804, -2.564160, -0.758425, 1.570796, 1.641921],accel_mss,speed_ms,0,blend_radius_m)
    |   movel([0.070507, -1.389824, -2.564145, -0.758420, 1.570796, 1.641303],accel_mss,speed_ms,0,blend_radius_m)
    |   movel([0.069879, -1.389788, -2.564171, -0.758430, 1.570796, 1.640675],accel_mss,speed_ms,0,blend_radius_m)
    |   movel([0.069421, -1.389680, -2.564249, -0.758460, 1.570796, 1.640217],accel_mss,speed_ms,0,blend_radius_m)
    |   movel([0.068816, -1.389330, -2.564501, -0.758558, 1.570796, 1.639612],accel_mss,speed_ms,0,blend_radius_m)
    |   movel([0.068448, -1.388813, -2.564872, -0.758704, 1.570796, 1.639245],accel_mss,speed_ms,0,blend_radius_m)
    |   movel([0.068281, -1.388058, -2.565413, -0.758917, 1.570796, 1.639078],accel_mss,speed_ms,0,blend_radius_m)
    |   movel([0.068297, -1.386960, -2.566200, -0.759229, 1.570796, 1.639093],accel_mss,speed_ms,0,blend_radius_m)
    |   movel([0.068504, -1.385834, -2.567004, -0.759551, 1.570796, 1.639300],accel_mss,speed_ms,0,blend_radius_m)
    |   movel([0.068940, -1.384856, -2.567702, -0.759832, 1.570796, 1.639736],accel_mss,speed_ms,0,blend_radius_m)
    |   movel([0.069611, -1.384023, -2.568295, -0.760072, 1.570796, 1.640407],accel_mss,speed_ms,0,blend_radius_m)
    |   movel([0.070503, -1.383332, -2.568785, -0.760272, 1.570796, 1.641299],accel_mss,speed_ms,0,blend_radius_m)
    |   movel([0.071108, -1.383026, -2.569002, -0.760360, 1.570796, 1.641904],accel_mss,speed_ms,0,blend_radius_m)
    |   movel([0.071382, -1.383068, -2.568972, -0.760348, 1.570796, 1.642178],accel_mss,speed_ms,0,blend_radius_m)
    |   movel([0.071487, -1.383440, -2.568708, -0.760240, 1.570796, 1.642283],accel_mss,speed_ms,0,blend_radius_m)
    |   movel([0.071463, -1.384769, -2.567763, -0.759856, 1.570796, 1.642260],accel_mss,speed_ms,0,blend_radius_m)
    |   movel([0.071447, -1.385513, -2.567233, -0.759643, 1.570796, 1.642243],accel_mss,speed_ms,0,blend_radius_m)
    |   movel([0.071447, -1.386326, -2.566653, -0.759410, 1.570796, 1.642243],accel_mss,speed_ms,0,blend_radius_m)
    |   movel([0.071456, -1.387087, -2.566109, -0.759193, 1.570796, 1.642252],accel_mss,speed_ms,0,blend_radius_m)
    |   movel([0.071478, -1.387656, -2.565702, -0.759031, 1.570796, 1.642275],accel_mss,speed_ms,0,blend_radius_m)
    |   movel([0.071526, -1.388621, -2.565010, -0.758758, 1.570796, 1.642322],accel_mss,speed_ms,0,blend_radius_m)
    |   movel([0.071525, -1.389181, -2.564608, -0.758600, 1.570796, 1.642321],accel_mss,speed_ms,0,blend_radius_m)
    |   movel([0.071490, -1.389540, -2.564349, -0.758499, 1.570796, 1.642286],accel_mss,speed_ms,0,blend_radius_m)
    |   speed_ms = 0.003
    |   movel([0.071390, -1.392961, -2.565710, -0.753718, 1.570796, 1.642186],accel_mss,speed_ms,0,blend_radius_m)
    |   speed_ms = 0.007
    |   movel([0.071125, -1.393071, -2.565630, -0.753687, 1.570796, 1.641921],accel_mss,speed_ms,0,blend_radius_m)
    |   movel([0.070507, -1.393091, -2.565616, -0.753682, 1.570796, 1.641303],accel_mss,speed_ms,0,blend_radius_m)
    |   movel([0.069879, -1.393055, -2.565642, -0.753692, 1.570796, 1.640675],accel_mss,speed_ms,0,blend_radius_m)
    |   movel([0.069421, -1.392947, -2.565720, -0.753722, 1.570796, 1.640217],accel_mss,speed_ms,0,blend_radius_m)
    |   movel([0.068816, -1.392599, -2.565972, -0.753819, 1.570796, 1.639612],accel_mss,speed_ms,0,blend_radius_m)
    |   movel([0.068448, -1.392083, -2.566344, -0.753962, 1.570796, 1.639245],accel_mss,speed_ms,0,blend_radius_m)
    |   movel([0.068281, -1.391330, -2.566887, -0.754172, 1.570796, 1.639078],accel_mss,speed_ms,0,blend_radius_m)
    |   movel([0.068297, -1.390235, -2.567675, -0.754479, 1.570796, 1.639093],accel_mss,speed_ms,0,blend_radius_m)
    |   movel([0.068504, -1.389112, -2.568481, -0.754795, 1.570796, 1.639300],accel_mss,speed_ms,0,blend_radius_m)
    |   movel([0.068940, -1.388136, -2.569181, -0.755072, 1.570796, 1.639736],accel_mss,speed_ms,0,blend_radius_m)
    |   movel([0.069611, -1.387306, -2.569775, -0.755309, 1.570796, 1.640407],accel_mss,speed_ms,0,blend_radius_m)
    |   movel([0.070503, -1.386617, -2.570266, -0.755506, 1.570796, 1.641299],accel_mss,speed_ms,0,blend_radius_m)
    |   movel([0.071108, -1.386312, -2.570484, -0.755593, 1.570796, 1.641904],accel_mss,speed_ms,0,blend_radius_m)
    |   movel([0.071382, -1.386354, -2.570454, -0.755581, 1.570796, 1.642178],accel_mss,speed_ms,0,blend_radius_m)
    |   movel([0.071487, -1.386725, -2.570189, -0.755475, 1.570796, 1.642283],accel_mss,speed_ms,0,blend_radius_m)
    |   movel([0.071463, -1.388050, -2.569242, -0.755097, 1.570796, 1.642260],accel_mss,speed_ms,0,blend_radius_m)
    |   movel([0.071447, -1.388792, -2.568711, -0.754886, 1.570796, 1.642243],accel_mss,speed_ms,0,blend_radius_m)
    |   movel([0.071447, -1.389603, -2.568129, -0.754657, 1.570796, 1.642243],accel_mss,speed_ms,0,blend_radius_m)
    |   movel([0.071456, -1.390362, -2.567584, -0.754443, 1.570796, 1.642252],accel_mss,speed_ms,0,blend_radius_m)
    |   movel([0.071478, -1.390929, -2.567176, -0.754284, 1.570796, 1.642275],accel_mss,speed_ms,0,blend_radius_m)
    |   movel([0.071526, -1.391892, -2.566482, -0.754015, 1.570796, 1.642322],accel_mss,speed_ms,0,blend_radius_m)
    |   movel([0.071525, -1.392450, -2.566079, -0.753860, 1.570796, 1.642321],accel_mss,speed_ms,0,blend_radius_m)
    |   movel([0.071490, -1.392808, -2.565821, -0.753760, 1.570796, 1.642286],accel_mss,speed_ms,0,blend_radius_m)
    |   speed_ms = 0.003
    |   movel([0.071390, -1.380023, -2.559776, -0.772590, 1.570796, 1.642186],accel_mss,speed_ms,0,blend_radius_m)
    |   speed_ms = 1.000
    |   movel([0.071390, -1.355193, -2.547515, -0.809680, 1.570796, 1.642186],accel_mss,speed_ms,0,blend_radius_m)
    |   movel([0.064153, -1.352173, -2.549573, -0.810644, 1.570796, 1.634949],accel_mss,speed_ms,0,blend_radius_m)
    |   movel([0.064153, -1.377057, -2.561872, -0.773460, 1.570796, 1.634949],accel_mss,speed_ms,0,blend_radius_m)
    |   speed_ms = 0.003
    |   movel([0.064153, -1.386751, -2.566349, -0.759289, 1.570796, 1.634949],accel_mss,speed_ms,0,blend_radius_m)
    |   speed_ms = 0.007
    |   movel([0.063340, -1.387772, -2.565619, -0.758999, 1.570796, 1.634136],accel_mss,speed_ms,0,blend_radius_m)
    |   movel([0.062686, -1.388569, -2.565047, -0.758773, 1.570796, 1.633482],accel_mss,speed_ms,0,blend_radius_m)
    |   movel([0.062675, -1.388124, -2.565366, -0.758899, 1.570796, 1.633471],accel_mss,speed_ms,0,blend_radius_m)
    |   movel([0.062900, -1.387745, -2.565638, -0.759006, 1.570796, 1.633696],accel_mss,speed_ms,0,blend_radius_m)
    |   movel([0.063169, -1.387429, -2.565864, -0.759096, 1.570796, 1.633965],accel_mss,speed_ms,0,blend_radius_m)
    |   movel([0.063443, -1.387047, -2.566137, -0.759204, 1.570796, 1.634239],accel_mss,speed_ms,0,blend_radius_m)
    |   movel([0.063524, -1.386809, -2.566308, -0.759272, 1.570796, 1.634320],accel_mss,speed_ms,0,blend_radius_m)
    |   movel([0.063593, -1.386471, -2.566549, -0.759368, 1.570796, 1.634389],accel_mss,speed_ms,0,blend_radius_m)
    |   movel([0.063654, -1.386177, -2.566759, -0.759452, 1.570796, 1.634450],accel_mss,speed_ms,0,blend_radius_m)
    |   movel([0.063753, -1.385826, -2.567010, -0.759553, 1.570796, 1.634549],accel_mss,speed_ms,0,blend_radius_m)
    |   movel([0.063869, -1.385475, -2.567261, -0.759654, 1.570796, 1.634666],accel_mss,speed_ms,0,blend_radius_m)
    |   movel([0.063989, -1.385181, -2.567470, -0.759738, 1.570796, 1.634785],accel_mss,speed_ms,0,blend_radius_m)
    |   movel([0.064155, -1.384750, -2.567777, -0.759862, 1.570796, 1.634951],accel_mss,speed_ms,0,blend_radius_m)
    |   movel([0.064180, -1.384485, -2.567966, -0.759938, 1.570796, 1.634976],accel_mss,speed_ms,0,blend_radius_m)
    |   movel([0.063844, -1.384381, -2.568040, -0.759968, 1.570796, 1.634641],accel_mss,speed_ms,0,blend_radius_m)
    |   movel([0.063665, -1.384201, -2.568168, -0.760020, 1.570796, 1.634461],accel_mss,speed_ms,0,blend_radius_m)
    |   movel([0.063664, -1.383761, -2.568481, -0.760147, 1.570796, 1.634460],accel_mss,speed_ms,0,blend_radius_m)
    |   movel([0.063663, -1.383539, -2.568639, -0.760212, 1.570796, 1.634460],accel_mss,speed_ms,0,blend_radius_m)
    |   movel([0.063659, -1.383178, -2.568894, -0.760316, 1.570796, 1.634455],accel_mss,speed_ms,0,blend_radius_m)
    |   movel([0.063652, -1.382770, -2.569184, -0.760435, 1.570796, 1.634449],accel_mss,speed_ms,0,blend_radius_m)
    |   movel([0.063644, -1.382363, -2.569473, -0.760553, 1.570796, 1.634440],accel_mss,speed_ms,0,blend_radius_m)
    |   movel([0.063647, -1.381532, -2.570061, -0.760796, 1.570796, 1.634444],accel_mss,speed_ms,0,blend_radius_m)
    |   movel([0.063692, -1.380836, -2.570553, -0.761000, 1.570796, 1.634488],accel_mss,speed_ms,0,blend_radius_m)
    |   movel([0.063775, -1.380285, -2.570942, -0.761162, 1.570796, 1.634571],accel_mss,speed_ms,0,blend_radius_m)
    |   movel([0.063897, -1.379969, -2.571165, -0.761255, 1.570796, 1.634693],accel_mss,speed_ms,0,blend_radius_m)
    |   movel([0.064290, -1.379690, -2.571361, -0.761337, 1.570796, 1.635086],accel_mss,speed_ms,0,blend_radius_m)
    |   movel([0.064739, -1.379526, -2.571477, -0.761386, 1.570796, 1.635535],accel_mss,speed_ms,0,blend_radius_m)
    |   movel([0.065708, -1.379220, -2.571693, -0.761476, 1.570796, 1.636505],accel_mss,speed_ms,0,blend_radius_m)
    |   movel([0.066539, -1.378970, -2.571869, -0.761550, 1.570796, 1.637335],accel_mss,speed_ms,0,blend_radius_m)
    |   movel([0.067034, -1.378840, -2.571960, -0.761589, 1.570796, 1.637831],accel_mss,speed_ms,0,blend_radius_m)
    |   movel([0.067345, -1.378784, -2.571999, -0.761605, 1.570796, 1.638141],accel_mss,speed_ms,0,blend_radius_m)
    |   movel([0.067187, -1.379390, -2.571573, -0.761426, 1.570796, 1.637983],accel_mss,speed_ms,0,blend_radius_m)
    |   movel([0.066879, -1.379944, -2.571182, -0.761262, 1.570796, 1.637675],accel_mss,speed_ms,0,blend_radius_m)
    |   movel([0.066506, -1.380579, -2.570734, -0.761075, 1.570796, 1.637303],accel_mss,speed_ms,0,blend_radius_m)
    |   movel([0.066134, -1.381213, -2.570286, -0.760889, 1.570796, 1.636931],accel_mss,speed_ms,0,blend_radius_m)
    |   movel([0.065832, -1.381769, -2.569893, -0.760727, 1.570796, 1.636628],accel_mss,speed_ms,0,blend_radius_m)
    |   movel([0.065596, -1.382232, -2.569566, -0.760592, 1.570796, 1.636392],accel_mss,speed_ms,0,blend_radius_m)
    |   movel([0.065843, -1.382380, -2.569460, -0.760548, 1.570796, 1.636640],accel_mss,speed_ms,0,blend_radius_m)
    |   movel([0.066139, -1.382317, -2.569505, -0.760567, 1.570796, 1.636935],accel_mss,speed_ms,0,blend_radius_m)
    |   movel([0.066626, -1.382174, -2.569607, -0.760609, 1.570796, 1.637423],accel_mss,speed_ms,0,blend_radius_m)
    |   movel([0.067199, -1.382006, -2.569725, -0.760657, 1.570796, 1.637995],accel_mss,speed_ms,0,blend_radius_m)
    |   movel([0.067529, -1.381937, -2.569775, -0.760678, 1.570796, 1.638325],accel_mss,speed_ms,0,blend_radius_m)
    |   movel([0.067763, -1.382007, -2.569725, -0.760657, 1.570796, 1.638559],accel_mss,speed_ms,0,blend_radius_m)
    |   movel([0.067012, -1.383013, -2.569012, -0.760364, 1.570796, 1.637808],accel_mss,speed_ms,0,blend_radius_m)
    |   movel([0.066191, -1.384094, -2.568244, -0.760051, 1.570796, 1.636988],accel_mss,speed_ms,0,blend_radius_m)
    |   movel([0.065221, -1.385365, -2.567339, -0.759685, 1.570796, 1.636018],accel_mss,speed_ms,0,blend_radius_m)
    |   movel([0.064153, -1.386751, -2.566349, -0.759289, 1.570796, 1.634949],accel_mss,speed_ms,0,blend_radius_m)
    |   speed_ms = 0.003
    |   movel([0.064153, -1.390026, -2.567825, -0.754538, 1.570796, 1.634949],accel_mss,speed_ms,0,blend_radius_m)
    |   speed_ms = 0.007
    |   movel([0.063340, -1.391044, -2.567093, -0.754252, 1.570796, 1.634136],accel_mss,speed_ms,0,blend_radius_m)
    |   movel([0.062686, -1.391840, -2.566520, -0.754030, 1.570796, 1.633482],accel_mss,speed_ms,0,blend_radius_m)
    |   movel([0.062675, -1.391396, -2.566839, -0.754153, 1.570796, 1.633471],accel_mss,speed_ms,0,blend_radius_m)
    |   movel([0.062900, -1.391018, -2.567112, -0.754259, 1.570796, 1.633696],accel_mss,speed_ms,0,blend_radius_m)
    |   movel([0.063169, -1.390703, -2.567339, -0.754348, 1.570796, 1.633965],accel_mss,speed_ms,0,blend_radius_m)
    |   movel([0.063443, -1.390322, -2.567612, -0.754454, 1.570796, 1.634239],accel_mss,speed_ms,0,blend_radius_m)
    |   movel([0.063524, -1.390085, -2.567783, -0.754521, 1.570796, 1.634320],accel_mss,speed_ms,0,blend_radius_m)
    |   movel([0.063593, -1.389748, -2.568025, -0.754616, 1.570796, 1.634389],accel_mss,speed_ms,0,blend_radius_m)
    |   movel([0.063654, -1.389454, -2.568236, -0.754699, 1.570796, 1.634450],accel_mss,speed_ms,0,blend_radius_m)
    |   movel([0.063753, -1.389104, -2.568487, -0.754798, 1.570796, 1.634549],accel_mss,speed_ms,0,blend_radius_m)
    |   movel([0.063869, -1.388754, -2.568738, -0.754897, 1.570796, 1.634666],accel_mss,speed_ms,0,blend_radius_m)
    |   movel([0.063989, -1.388461, -2.568948, -0.754980, 1.570796, 1.634785],accel_mss,speed_ms,0,blend_radius_m)
    |   movel([0.064155, -1.388031, -2.569256, -0.755102, 1.570796, 1.634951],accel_mss,speed_ms,0,blend_radius_m)
    |   movel([0.064180, -1.387767, -2.569445, -0.755177, 1.570796, 1.634976],accel_mss,speed_ms,0,blend_radius_m)
    |   movel([0.063844, -1.387663, -2.569519, -0.755207, 1.570796, 1.634641],accel_mss,speed_ms,0,blend_radius_m)
    |   movel([0.063665, -1.387484, -2.569647, -0.755258, 1.570796, 1.634461],accel_mss,speed_ms,0,blend_radius_m)
    |   movel([0.063664, -1.387045, -2.569961, -0.755383, 1.570796, 1.634460],accel_mss,speed_ms,0,blend_radius_m)
    |   movel([0.063663, -1.386823, -2.570119, -0.755447, 1.570796, 1.634460],accel_mss,speed_ms,0,blend_radius_m)
    |   movel([0.063659, -1.386464, -2.570376, -0.755550, 1.570796, 1.634455],accel_mss,speed_ms,0,blend_radius_m)
    |   movel([0.063652, -1.386057, -2.570666, -0.755666, 1.570796, 1.634449],accel_mss,speed_ms,0,blend_radius_m)
    |   movel([0.063644, -1.385650, -2.570956, -0.755783, 1.570796, 1.634440],accel_mss,speed_ms,0,blend_radius_m)
    |   movel([0.063647, -1.384822, -2.571545, -0.756022, 1.570796, 1.634444],accel_mss,speed_ms,0,blend_radius_m)
    |   movel([0.063692, -1.384128, -2.572038, -0.756223, 1.570796, 1.634488],accel_mss,speed_ms,0,blend_radius_m)
    |   movel([0.063775, -1.383578, -2.572429, -0.756383, 1.570796, 1.634571],accel_mss,speed_ms,0,blend_radius_m)
    |   movel([0.063897, -1.383263, -2.572652, -0.756474, 1.570796, 1.634693],accel_mss,speed_ms,0,blend_radius_m)
    |   movel([0.064290, -1.382985, -2.572849, -0.756555, 1.570796, 1.635086],accel_mss,speed_ms,0,blend_radius_m)
    |   movel([0.064739, -1.382821, -2.572964, -0.756603, 1.570796, 1.635535],accel_mss,speed_ms,0,blend_radius_m)
    |   movel([0.065708, -1.382516, -2.573181, -0.756692, 1.570796, 1.636505],accel_mss,speed_ms,0,blend_radius_m)
    |   movel([0.066539, -1.382267, -2.573357, -0.756765, 1.570796, 1.637335],accel_mss,speed_ms,0,blend_radius_m)
    |   movel([0.067034, -1.382137, -2.573449, -0.756803, 1.570796, 1.637831],accel_mss,speed_ms,0,blend_radius_m)
    |   movel([0.067345, -1.382082, -2.573488, -0.756819, 1.570796, 1.638141],accel_mss,speed_ms,0,blend_radius_m)
    |   movel([0.067187, -1.382685, -2.573061, -0.756643, 1.570796, 1.637983],accel_mss,speed_ms,0,blend_radius_m)
    |   movel([0.066879, -1.383239, -2.572669, -0.756481, 1.570796, 1.637675],accel_mss,speed_ms,0,blend_radius_m)
    |   movel([0.066506, -1.383872, -2.572220, -0.756297, 1.570796, 1.637303],accel_mss,speed_ms,0,blend_radius_m)
    |   movel([0.066134, -1.384504, -2.571771, -0.756114, 1.570796, 1.636931],accel_mss,speed_ms,0,blend_radius_m)
    |   movel([0.065832, -1.385059, -2.571377, -0.755954, 1.570796, 1.636628],accel_mss,speed_ms,0,blend_radius_m)
    |   movel([0.065596, -1.385520, -2.571049, -0.755821, 1.570796, 1.636392],accel_mss,speed_ms,0,blend_radius_m)
    |   movel([0.065843, -1.385668, -2.570943, -0.755778, 1.570796, 1.636640],accel_mss,speed_ms,0,blend_radius_m)
    |   movel([0.066139, -1.385605, -2.570988, -0.755796, 1.570796, 1.636935],accel_mss,speed_ms,0,blend_radius_m)
    |   movel([0.066626, -1.385462, -2.571090, -0.755837, 1.570796, 1.637423],accel_mss,speed_ms,0,blend_radius_m)
    |   movel([0.067199, -1.385295, -2.571209, -0.755885, 1.570796, 1.637995],accel_mss,speed_ms,0,blend_radius_m)
    |   movel([0.067529, -1.385225, -2.571258, -0.755906, 1.570796, 1.638325],accel_mss,speed_ms,0,blend_radius_m)
    |   movel([0.067763, -1.385295, -2.571208, -0.755885, 1.570796, 1.638559],accel_mss,speed_ms,0,blend_radius_m)
    |   movel([0.067012, -1.386299, -2.570493, -0.755597, 1.570796, 1.637808],accel_mss,speed_ms,0,blend_radius_m)
    |   movel([0.066191, -1.387377, -2.569724, -0.755288, 1.570796, 1.636988],accel_mss,speed_ms,0,blend_radius_m)
    |   movel([0.065221, -1.388644, -2.568817, -0.754928, 1.570796, 1.636018],accel_mss,speed_ms,0,blend_radius_m)
    |   movel([0.064153, -1.390026, -2.567825, -0.754538, 1.570796, 1.634949],accel_mss,speed_ms,0,blend_radius_m)
    |   speed_ms = 0.003
    |   movel([0.064153, -1.377057, -2.561872, -0.773460, 1.570796, 1.634949],accel_mss,speed_ms,0,blend_radius_m)
    |   speed_ms = 1.000
    |   movel([0.064153, -1.352173, -2.549573, -0.810644, 1.570796, 1.634949],accel_mss,speed_ms,0,blend_radius_m)
    |   movel([0.065962, -1.340154, -2.557638, -0.814597, 1.570796, 1.636759],accel_mss,speed_ms,0,blend_radius_m)
    |   movel([0.065962, -1.365252, -2.570091, -0.777046, 1.570796, 1.636759],accel_mss,speed_ms,0,blend_radius_m)
    |   speed_ms = 0.003
    |   movel([0.065962, -1.375037, -2.574625, -0.762726, 1.570796, 1.636759],accel_mss,speed_ms,0,blend_radius_m)
    |   speed_ms = 0.007
    |   movel([0.065737, -1.374802, -2.574789, -0.762797, 1.570796, 1.636533],accel_mss,speed_ms,0,blend_radius_m)
    |   movel([0.065748, -1.374108, -2.575274, -0.763008, 1.570796, 1.636545],accel_mss,speed_ms,0,blend_radius_m)
    |   movel([0.065782, -1.373380, -2.575780, -0.763229, 1.570796, 1.636578],accel_mss,speed_ms,0,blend_radius_m)
    |   movel([0.066186, -1.373075, -2.575992, -0.763321, 1.570796, 1.636982],accel_mss,speed_ms,0,blend_radius_m)
    |   movel([0.067252, -1.372821, -2.576169, -0.763399, 1.570796, 1.638048],accel_mss,speed_ms,0,blend_radius_m)
    |   movel([0.068316, -1.372596, -2.576325, -0.763467, 1.570796, 1.639113],accel_mss,speed_ms,0,blend_radius_m)
    |   movel([0.068585, -1.372629, -2.576302, -0.763457, 1.570796, 1.639381],accel_mss,speed_ms,0,blend_radius_m)
    |   movel([0.068684, -1.372934, -2.576090, -0.763364, 1.570796, 1.639480],accel_mss,speed_ms,0,blend_radius_m)
    |   movel([0.068626, -1.373256, -2.575866, -0.763266, 1.570796, 1.639422],accel_mss,speed_ms,0,blend_radius_m)
    |   movel([0.068470, -1.373815, -2.575478, -0.763096, 1.570796, 1.639267],accel_mss,speed_ms,0,blend_radius_m)
    |   movel([0.068277, -1.374079, -2.575293, -0.763016, 1.570796, 1.639073],accel_mss,speed_ms,0,blend_radius_m)
    |   movel([0.067750, -1.374381, -2.575083, -0.762925, 1.570796, 1.638546],accel_mss,speed_ms,0,blend_radius_m)
    |   movel([0.067148, -1.374646, -2.574898, -0.762845, 1.570796, 1.637944],accel_mss,speed_ms,0,blend_radius_m)
    |   movel([0.066517, -1.374873, -2.574740, -0.762776, 1.570796, 1.637313],accel_mss,speed_ms,0,blend_radius_m)
    |   movel([0.065962, -1.375037, -2.574625, -0.762726, 1.570796, 1.636759],accel_mss,speed_ms,0,blend_radius_m)
    |   speed_ms = 0.003
